KUKA KRL program: PPR-top-01.src

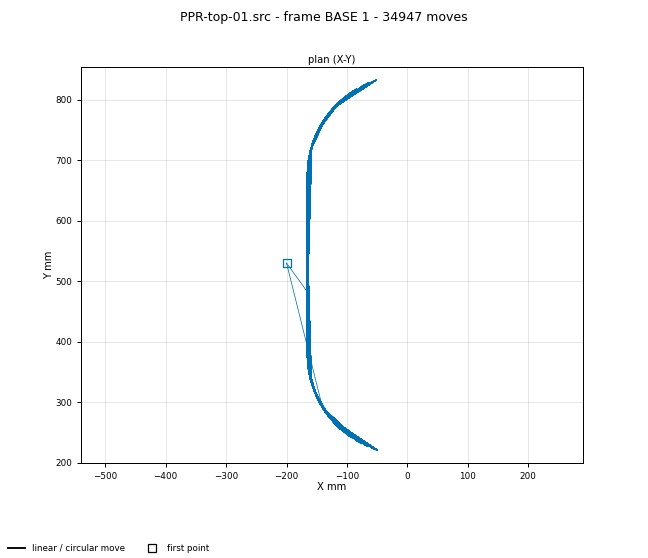
[picture p0: tool path of PPR-top-01.src in frame BASE 1, 34947 of 34948 moves have a stored position in this frame; points joined in program order, loops and branches not executed]
&ACCESS RVEO
&REL 11
&PARAM TEMPLATE = C:\KRC\Roboter\Template\vorgabe
&PARAM EDITMASK = *
DEF variable_helical2( )
;FOLD INI
  ;FOLD BASISTECH INI
    GLOBAL INTERRUPT DECL 3 WHEN $STOPMESS==TRUE DO IR_STOPM ( )
    INTERRUPT ON 3
    BAS (#INITMOV,0 )
  ;ENDFOLD (BASISTECH INI)
 ;FOLD USER INI


    ;Make your modifications here
  ;ENDFOLD (USER INI)
;ENDFOLD (INI)
ACTION(#AXIS_RESET,34,1000,#NOERROR,ERROR_CODE)
;FOLD PTP HOME  Vel= 100 % DEFAULT;%{PE}%MKUKATPBASIS,%CMOVE,%VPTP,%P 1:PTP, 2:HOME, 3:, 5:100, 7:DEFAULT
$BWDSTART = FALSE
PDAT_ACT=PDEFAULT
FDAT_ACT=FHOME
BAS (#PTP_PARAMS,100 )
$H_POS=XHOME
PTP  XHOME
;ENDFOLD
BAS(#TOOL,1)
BAS(#BASE,1)
$VEL_AXIS[1]=100
$VEL_AXIS[2]=100
$VEL_AXIS[3]=100
$VEL_AXIS[4]=100
$VEL_AXIS[5]=100
$VEL_AXIS[6]=100
$VEL_EXTAX[1]=100
$VEL_EXTAX[2]=100

$ACC_AXIS[1]=100
$ACC_AXIS[2]=100
$ACC_AXIS[3]=100
$ACC_AXIS[4]=100
$ACC_AXIS[5]=100
$ACC_AXIS[6]=100
$ACC_EXTAX[1]=100
$ACC_EXTAX[2]=100

;;;;;;;;; postprocessing parameters (date 2024-01-25T18:15:35.064605)
; qxconst: -165.65
; qxconstarcys: -151.5,145.5
; qE3offset: 0.00
; qyoffset: 530.00
; qswitchsplit: 3
; qthinningtol: 0.2010
;;;;;;;;;

SLIN {X  -200.000, Y  +530.000, Z    +0.000, A    +0.000, E1    +0.000, E3    +0.000, E4    +0.000}

SLIN {X  -140.419, Y  +290.622, Z    +0.000, E1   +73.705, E3  +372.898}
HALT
SPLINE
SPL {X  -135.839, Y  +283.697, Z    +0.000, E1   +73.388, E3  +378.636}
SPL {X  -131.903, Y  +278.292, Z    +0.000, E1   +73.096, E3  +383.125}
SPL {X  -129.007, Y  +274.590, Z    +0.000, E1   +72.484, E3  +388.421}
SPL {X  -124.646, Y  +269.397, Z    +0.000, E1   +72.041, E3  +393.170}
SPL {X  -111.023, Y  +255.562, Z    +0.000, E1   +75.772, E3  +384.951}
SPL {X   -49.289, Y  +220.353, Z    +0.000, E1   +56.690, E3  +577.666}
ENDSPLINE

SPLINE
SPL {X  -127.117, Y  +272.287, Z    +0.000, E1   +62.713, E3  +746.888}
SPL {X  -152.442, Y  +313.682, Z    +0.000, E1   +51.943, E3  +751.120}
SPL {X  -159.925, Y  +335.326, Z    +0.000, E1   +41.361, E3  +751.062}
SPL {X  -163.450, Y  +351.595, Z    +0.000, E1   +29.785, E3  +750.173}
SPL {X  -165.127, Y  +365.342, Z    +0.000, E1   +17.250, E3  +750.153}
SPL {X  -165.640, Y  +376.693, Z    +0.000, E1    +4.721, E3  +749.726}
SPL {X  -165.650, Y  +380.500, Z    +0.000, E1    -0.000, E3  +748.877}
SPL {X  -165.650, Y  +382.123, Z    +0.000, E1    -3.912, E3  +748.504}
SPL {X  -165.650, Y  +387.069, Z    +0.000, E1   -17.420, E3  +748.216}
SPL {X  -165.650, Y  +393.439, Z    +0.000, E1   -35.398, E3  +747.762}
SPL {X  -165.650, Y  +400.610, Z    +0.000, E1   -50.510, E3  +747.499}
SPL {X  -165.650, Y  +414.376, Z    +0.000, E1   -68.098, E3  +745.533}
SPL {X  -165.650, Y  +468.582, Z    +0.000, E1   -78.237, E3  +754.303}
SPL {X  -160.244, Y  +717.475, Z    +0.000, E1   -78.917, E3  +826.861}
SPL {X  -159.651, Y  +719.676, Z    +0.000, E1   -75.661, E3  +863.248}
SPL {X  -157.156, Y  +727.862, Z    +0.000, E1   -75.175, E3  +872.730}
SPL {X  -152.814, Y  +739.436, Z    +0.000, E1   -74.813, E3  +882.583}
SPL {X  -148.754, Y  +748.385, Z    +0.000, E1   -74.281, E3  +892.026}
SPL {X  -144.163, Y  +757.090, Z    +0.000, E1   -74.033, E3  +898.685}
SPL {X  -140.473, Y  +763.291, Z    +0.000, E1   -73.478, E3  +906.126}
SPL {X  -135.914, Y  +770.196, Z    +0.000, E1   -72.974, E3  +913.302}
SPL {X  -131.459, Y  +776.289, Z    +0.000, E1   -72.475, E3  +919.378}
SPL {X  -128.771, Y  +779.702, Z    +0.000, E1   -71.875, E3  +924.325}
SPL {X  -125.267, Y  +783.889, Z    +0.000, E1   -71.674, E3  +927.437}
SPL {X  -119.086, Y  +790.645, Z    +0.000, E1   -72.931, E3  +925.724}
SPL {X   -51.449, Y  +832.958, Z    +0.000, E1   -57.230, E3 +1083.244}
ENDSPLINE

SPLINE
SPL {X  -123.821, Y  +785.537, Z    +0.000, E1   -64.536, E3 +1284.989}
SPL {X  -153.467, Y  +737.853, Z    +0.000, E1   -51.757, E3 +1287.304}
SPL {X  -161.000, Y  +714.475, Z    +0.000, E1   -39.424, E3 +1286.776}
SPL {X  -164.534, Y  +694.695, Z    +0.000, E1   -23.511, E3 +1285.066}
SPL {X  -165.597, Y  +679.703, Z    +0.000, E1    -7.645, E3 +1284.942}
SPL {X  -165.650, Y  +673.520, Z    +0.000, E1    -0.048, E3 +1283.894}
SPL {X  -165.650, Y  +671.692, Z    +0.000, E1    +4.450, E3 +1283.460}
SPL {X  -165.650, Y  +667.743, Z    +0.000, E1   +15.617, E3 +1283.378}
SPL {X  -165.650, Y  +662.891, Z    +0.000, E1   +29.740, E3 +1282.896}
SPL {X  -165.650, Y  +655.319, Z    +0.000, E1   +47.265, E3 +1282.745}
SPL {X  -165.650, Y  +642.000, Z    +0.000, E1   +65.561, E3 +1281.726}
SPL {X  -165.650, Y  +619.979, Z    +0.000, E1   +79.465, E3 +1277.733}
SPL {X  -165.650, Y  +569.632, Z    +0.000, E1   +78.783, E3 +1293.011}
SPL {X  -158.840, Y  +331.491, Z    +0.000, E1   +77.462, E3 +1379.322}
ENDSPLINE

SPLINE
SPL {X  -159.893, Y  +335.208, Z    +0.000, E1   +75.483, E3 +1400.056}
ENDSPLINE

SPLINE
SPL {X  -156.487, Y  +324.170, Z    +0.000, E1   +75.150, E3 +1409.437}
SPL {X  -142.256, Y  +293.629, Z    +0.000, E1   +77.020, E3 +1404.537}
ENDSPLINE

SPLINE
SPL {X  -142.811, Y  +294.566, Z    +0.000, E1   +75.668, E3 +1416.499}
ENDSPLINE

SPLINE
SPL {X  -141.646, Y  +292.615, Z    +0.000, E1   +74.702, E3 +1425.593}
SPL {X  -140.419, Y  +290.622, Z    +0.000, E1   +73.705, E3 +1434.436}
SPL {X  -135.839, Y  +283.697, Z    +0.000, E1   +73.388, E3 +1440.174}
SPL {X  -131.336, Y  +277.551, Z    +0.000, E1   +72.879, E3 +1446.427}
SPL {X  -126.848, Y  +271.966, Z    +0.000, E1   +72.322, E3 +1452.155}
SPL {X  -123.729, Y  +268.359, Z    +0.000, E1   +71.932, E3 +1455.624}
SPL {X  -111.023, Y  +255.562, Z    +0.000, E1   +75.772, E3 +1446.490}
SPL {X   -52.752, Y  +221.474, Z    +0.000, E1   +59.157, E3 +1575.741}
SPL {X   -49.901, Y  +220.545, Z    +0.000, E1   +56.696, E3 +1662.134}
ENDSPLINE

SPLINE
SPL {X  -127.117, Y  +272.287, Z    +0.000, E1   +62.713, E3 +1808.427}
SPL {X  -152.442, Y  +313.682, Z    +0.000, E1   +51.943, E3 +1812.658}
SPL {X  -162.319, Y  +345.447, Z    +0.000, E1   +34.671, E3 +1812.084}
SPL {X  -165.127, Y  +365.342, Z    +0.000, E1   +17.250, E3 +1811.692}
SPL {X  -165.640, Y  +376.693, Z    +0.000, E1    +4.721, E3 +1811.265}
SPL {X  -165.650, Y  +380.500, Z    +0.000, E1    -0.000, E3 +1810.416}
SPL {X  -165.650, Y  +383.262, Z    +0.000, E1    -6.645, E3 +1809.945}
SPL {X  -165.650, Y  +388.390, Z    +0.000, E1   -21.508, E3 +1809.733}
SPL {X  -165.650, Y  +393.439, Z    +0.000, E1   -35.398, E3 +1809.300}
SPL {X  -165.650, Y  +400.610, Z    +0.000, E1   -50.510, E3 +1809.038}
SPL {X  -165.650, Y  +414.376, Z    +0.000, E1   -68.098, E3 +1807.071}
SPL {X  -165.650, Y  +468.582, Z    +0.000, E1   -78.237, E3 +1815.841}
SPL {X  -158.306, Y  +724.277, Z    +0.000, E1   -77.461, E3 +1906.283}
ENDSPLINE

SPLINE
SPL {X  -160.145, Y  +717.851, Z    +0.000, E1   -75.386, E3 +1926.796}
ENDSPLINE

SPLINE
SPL {X  -157.156, Y  +727.862, Z    +0.000, E1   -75.175, E3 +1934.268}
SPL {X  -154.068, Y  +736.353, Z    +0.000, E1   -74.906, E3 +1941.443}
SPL {X  -149.738, Y  +746.340, Z    +0.000, E1   -74.451, E3 +1951.131}
SPL {X  -144.163, Y  +757.090, Z    +0.000, E1   -74.033, E3 +1960.223}
SPL {X  -139.284, Y  +765.165, Z    +0.000, E1   -73.322, E3 +1969.918}
SPL {X  -134.662, Y  +771.969, Z    +0.000, E1   -72.884, E3 +1976.249}
SPL {X  -131.459, Y  +776.289, Z    +0.000, E1   -72.475, E3 +1980.917}
SPL {X  -127.605, Y  +781.126, Z    +0.000, E1   -71.922, E3 +1986.361}
SPL {X  -124.773, Y  +784.457, Z    +0.000, E1   -71.383, E3 +1990.408}
SPL {X  -119.086, Y  +790.645, Z    +0.000, E1   -72.931, E3 +1987.262}
SPL {X   -54.274, Y  +832.006, Z    +0.000, E1   -58.502, E3 +2117.475}
SPL {X   -50.797, Y  +833.169, Z    +0.000, E1   -57.000, E3 +2212.824}
ENDSPLINE

SPLINE
SPL {X  -113.713, Y  +795.955, Z    +0.000, E1   -65.735, E3 +2343.701}
SPL {X  -131.116, Y  +776.736, Z    +0.000, E1   -63.149, E3 +2348.231}
SPL {X  -153.467, Y  +737.853, Z    +0.000, E1   -51.757, E3 +2348.842}
SPL {X  -162.176, Y  +709.248, Z    +0.000, E1   -35.773, E3 +2347.868}
SPL {X  -164.888, Y  +691.368, Z    +0.000, E1   -20.174, E3 +2346.305}
SPL {X  -165.597, Y  +679.703, Z    +0.000, E1    -7.645, E3 +2346.480}
SPL {X  -165.650, Y  +673.520, Z    +0.000, E1    -0.048, E3 +2345.432}
SPL {X  -165.650, Y  +671.692, Z    +0.000, E1    +4.450, E3 +2344.999}
SPL {X  -165.650, Y  +667.743, Z    +0.000, E1   +15.617, E3 +2344.917}
SPL {X  -165.650, Y  +662.891, Z    +0.000, E1   +29.740, E3 +2344.434}
SPL {X  -165.650, Y  +658.373, Z    +0.000, E1   +40.877, E3 +2344.632}
SPL {X  -165.650, Y  +650.834, Z    +0.000, E1   +55.143, E3 +2343.885}
SPL {X  -165.650, Y  +639.785, Z    +0.000, E1   +67.512, E3 +2343.102}
SPL {X  -165.650, Y  +619.979, Z    +0.000, E1   +79.465, E3 +2339.271}
SPL {X  -165.650, Y  +584.722, Z    +0.000, E1   +79.551, E3 +2348.562}
SPL {X  -165.650, Y  +560.326, Z    +0.000, E1   +78.360, E3 +2358.284}
SPL {X  -160.258, Y  +336.579, Z    +0.000, E1   +78.314, E3 +2429.806}
SPL {X  -159.618, Y  +334.207, Z    +0.000, E1   +75.622, E3 +2460.620}
SPL {X  -156.487, Y  +324.170, Z    +0.000, E1   +75.150, E3 +2470.976}
SPL {X  -142.256, Y  +293.629, Z    +0.000, E1   +77.020, E3 +2466.076}
ENDSPLINE

SPLINE
SPL {X  -142.811, Y  +294.566, Z    +0.000, E1   +75.668, E3 +2478.038}
ENDSPLINE

SPLINE
SPL {X  -141.646, Y  +292.615, Z    +0.000, E1   +74.702, E3 +2487.131}
SPL {X  -140.419, Y  +290.622, Z    +0.000, E1   +73.705, E3 +2495.975}
SPL {X  -136.008, Y  +283.940, Z    +0.000, E1   +73.594, E3 +2500.094}
SPL {X  -132.748, Y  +279.415, Z    +0.000, E1   +73.006, E3 +2506.150}
SPL {X  -129.007, Y  +274.590, Z    +0.000, E1   +72.484, E3 +2511.498}
SPL {X  -125.914, Y  +270.864, Z    +0.000, E1   +72.144, E3 +2514.990}
SPL {X  -123.729, Y  +268.359, Z    +0.000, E1   +71.932, E3 +2517.162}
SPL {X  -111.023, Y  +255.562, Z    +0.000, E1   +75.772, E3 +2508.028}
SPL {X   -49.289, Y  +220.353, Z    +0.000, E1   +56.690, E3 +2700.743}
ENDSPLINE

SPLINE
SPL {X  -127.117, Y  +272.287, Z    +0.000, E1   +62.713, E3 +2869.965}
SPL {X  -154.956, Y  +319.945, Z    +0.000, E1   +49.402, E3 +2874.364}
SPL {X  -162.871, Y  +348.286, Z    +0.000, E1   +32.462, E3 +2873.392}
SPL {X  -165.127, Y  +365.342, Z    +0.000, E1   +17.250, E3 +2873.230}
SPL {X  -165.640, Y  +376.693, Z    +0.000, E1    +4.721, E3 +2872.803}
SPL {X  -165.650, Y  +380.500, Z    +0.000, E1    -0.000, E3 +2871.954}
SPL {X  -165.650, Y  +382.123, Z    +0.000, E1    -3.912, E3 +2871.581}
SPL {X  -165.650, Y  +387.069, Z    +0.000, E1   -17.420, E3 +2871.293}
SPL {X  -165.650, Y  +393.439, Z    +0.000, E1   -35.398, E3 +2870.839}
SPL {X  -165.650, Y  +400.610, Z    +0.000, E1   -50.510, E3 +2870.576}
SPL {X  -165.650, Y  +414.376, Z    +0.000, E1   -68.098, E3 +2868.610}
SPL {X  -165.650, Y  +468.582, Z    +0.000, E1   -78.237, E3 +2877.380}
SPL {X  -160.244, Y  +717.475, Z    +0.000, E1   -78.917, E3 +2949.938}
SPL {X  -159.651, Y  +719.676, Z    +0.000, E1   -75.661, E3 +2986.324}
SPL {X  -157.156, Y  +727.862, Z    +0.000, E1   -75.175, E3 +2995.807}
SPL {X  -154.068, Y  +736.353, Z    +0.000, E1   -74.906, E3 +3002.981}
SPL {X  -149.738, Y  +746.340, Z    +0.000, E1   -74.451, E3 +3012.669}
SPL {X  -144.163, Y  +757.090, Z    +0.000, E1   -74.033, E3 +3021.762}
SPL {X  -139.284, Y  +765.165, Z    +0.000, E1   -73.322, E3 +3031.456}
SPL {X  -134.662, Y  +771.969, Z    +0.000, E1   -72.884, E3 +3037.788}
SPL {X  -131.459, Y  +776.289, Z    +0.000, E1   -72.475, E3 +3042.455}
SPL {X  -127.605, Y  +781.126, Z    +0.000, E1   -71.922, E3 +3047.899}
SPL {X  -124.773, Y  +784.457, Z    +0.000, E1   -71.383, E3 +3051.947}
SPL {X  -119.086, Y  +790.645, Z    +0.000, E1   -72.931, E3 +3048.801}
SPL {X   -51.449, Y  +832.958, Z    +0.000, E1   -57.230, E3 +3206.321}
ENDSPLINE

SPLINE
SPL {X  -123.821, Y  +785.537, Z    +0.000, E1   -64.536, E3 +3408.066}
SPL {X  -153.467, Y  +737.853, Z    +0.000, E1   -51.757, E3 +3410.381}
SPL {X  -161.000, Y  +714.475, Z    +0.000, E1   -39.424, E3 +3409.853}
SPL {X  -164.534, Y  +694.695, Z    +0.000, E1   -23.511, E3 +3408.143}
SPL {X  -165.597, Y  +679.703, Z    +0.000, E1    -7.645, E3 +3408.019}
SPL {X  -165.650, Y  +673.520, Z    +0.000, E1    -0.048, E3 +3406.971}
SPL {X  -165.650, Y  +671.692, Z    +0.000, E1    +4.450, E3 +3406.537}
SPL {X  -165.650, Y  +667.743, Z    +0.000, E1   +15.617, E3 +3406.455}
SPL {X  -165.650, Y  +661.459, Z    +0.000, E1   +33.218, E3 +3406.035}
SPL {X  -165.650, Y  +653.296, Z    +0.000, E1   +51.333, E3 +3405.591}
SPL {X  -165.650, Y  +642.000, Z    +0.000, E1   +65.561, E3 +3404.803}
SPL {X  -165.650, Y  +619.979, Z    +0.000, E1   +79.465, E3 +3400.810}
SPL {X  -165.650, Y  +569.632, Z    +0.000, E1   +78.783, E3 +3416.088}
SPL {X  -158.840, Y  +331.491, Z    +0.000, E1   +77.462, E3 +3502.398}
ENDSPLINE

SPLINE
SPL {X  -159.893, Y  +335.208, Z    +0.000, E1   +75.483, E3 +3523.133}
ENDSPLINE

SPLINE
SPL {X  -156.487, Y  +324.170, Z    +0.000, E1   +75.150, E3 +3532.514}
SPL {X  -142.256, Y  +293.629, Z    +0.000, E1   +77.020, E3 +3527.614}
ENDSPLINE

SPLINE
SPL {X  -142.811, Y  +294.566, Z    +0.000, E1   +75.668, E3 +3539.576}
ENDSPLINE

SPLINE
SPL {X  -141.646, Y  +292.615, Z    +0.000, E1   +74.702, E3 +3548.670}
SPL {X  -140.419, Y  +290.622, Z    +0.000, E1   +73.705, E3 +3557.513}
SPL {X  -136.008, Y  +283.940, Z    +0.000, E1   +73.594, E3 +3561.632}
SPL {X  -132.748, Y  +279.415, Z    +0.000, E1   +73.006, E3 +3567.688}
SPL {X  -129.007, Y  +274.590, Z    +0.000, E1   +72.484, E3 +3573.037}
SPL {X  -125.914, Y  +270.864, Z    +0.000, E1   +72.144, E3 +3576.528}
SPL {X  -123.729, Y  +268.359, Z    +0.000, E1   +71.932, E3 +3578.701}
SPL {X  -111.023, Y  +255.562, Z    +0.000, E1   +75.772, E3 +3569.567}
SPL {X   -49.289, Y  +220.353, Z    +0.000, E1   +56.690, E3 +3762.282}
ENDSPLINE

SPLINE
SPL {X  -127.117, Y  +272.287, Z    +0.000, E1   +62.713, E3 +3931.503}
SPL {X  -154.956, Y  +319.945, Z    +0.000, E1   +49.402, E3 +3935.903}
SPL {X  -162.871, Y  +348.286, Z    +0.000, E1   +32.462, E3 +3934.930}
SPL {X  -165.127, Y  +365.342, Z    +0.000, E1   +17.250, E3 +3934.769}
SPL {X  -165.640, Y  +376.693, Z    +0.000, E1    +4.721, E3 +3934.342}
SPL {X  -165.650, Y  +380.500, Z    +0.000, E1    -0.000, E3 +3933.493}
SPL {X  -165.650, Y  +383.262, Z    +0.000, E1    -6.645, E3 +3933.022}
SPL {X  -165.650, Y  +388.390, Z    +0.000, E1   -21.508, E3 +3932.809}
SPL {X  -165.650, Y  +393.439, Z    +0.000, E1   -35.398, E3 +3932.377}
SPL {X  -165.650, Y  +400.610, Z    +0.000, E1   -50.510, E3 +3932.115}
SPL {X  -165.650, Y  +414.376, Z    +0.000, E1   -68.098, E3 +3930.148}
SPL {X  -165.650, Y  +468.582, Z    +0.000, E1   -78.237, E3 +3938.918}
SPL {X  -158.306, Y  +724.277, Z    +0.000, E1   -77.461, E3 +4029.360}
ENDSPLINE

SPLINE
SPL {X  -160.145, Y  +717.851, Z    +0.000, E1   -75.386, E3 +4049.873}
ENDSPLINE

SPLINE
SPL {X  -157.156, Y  +727.862, Z    +0.000, E1   -75.175, E3 +4057.345}
SPL {X  -154.068, Y  +736.353, Z    +0.000, E1   -74.906, E3 +4064.520}
SPL {X  -149.738, Y  +746.340, Z    +0.000, E1   -74.451, E3 +4074.208}
SPL {X  -144.163, Y  +757.090, Z    +0.000, E1   -74.033, E3 +4083.300}
SPL {X  -139.284, Y  +765.165, Z    +0.000, E1   -73.322, E3 +4092.995}
SPL {X  -134.662, Y  +771.969, Z    +0.000, E1   -72.884, E3 +4099.326}
SPL {X  -131.459, Y  +776.289, Z    +0.000, E1   -72.475, E3 +4103.994}
SPL {X  -127.605, Y  +781.126, Z    +0.000, E1   -71.922, E3 +4109.438}
SPL {X  -124.773, Y  +784.457, Z    +0.000, E1   -71.383, E3 +4113.485}
SPL {X  -119.086, Y  +790.645, Z    +0.000, E1   -72.931, E3 +4110.339}
SPL {X   -51.449, Y  +832.958, Z    +0.000, E1   -57.230, E3 +4267.859}
ENDSPLINE

SPLINE
SPL {X  -123.821, Y  +785.537, Z    +0.000, E1   -64.536, E3 +4469.604}
SPL {X  -153.467, Y  +737.853, Z    +0.000, E1   -51.757, E3 +4471.919}
SPL {X  -161.000, Y  +714.475, Z    +0.000, E1   -39.424, E3 +4471.392}
SPL {X  -164.534, Y  +694.695, Z    +0.000, E1   -23.511, E3 +4469.682}
SPL {X  -165.597, Y  +679.703, Z    +0.000, E1    -7.645, E3 +4469.557}
SPL {X  -165.650, Y  +673.520, Z    +0.000, E1    -0.048, E3 +4468.509}
SPL {X  -165.650, Y  +671.692, Z    +0.000, E1    +4.450, E3 +4468.076}
SPL {X  -165.650, Y  +667.743, Z    +0.000, E1   +15.617, E3 +4467.994}
SPL {X  -165.650, Y  +661.459, Z    +0.000, E1   +33.218, E3 +4467.574}
SPL {X  -165.650, Y  +653.296, Z    +0.000, E1   +51.333, E3 +4467.129}
SPL {X  -165.650, Y  +642.000, Z    +0.000, E1   +65.561, E3 +4466.341}
SPL {X  -165.650, Y  +619.979, Z    +0.000, E1   +79.465, E3 +4462.348}
SPL {X  -165.650, Y  +569.632, Z    +0.000, E1   +78.783, E3 +4477.627}
SPL {X  -158.840, Y  +331.491, Z    +0.000, E1   +77.462, E3 +4563.937}
ENDSPLINE

SPLINE
SPL {X  -159.893, Y  +335.208, Z    +0.000, E1   +75.483, E3 +4584.672}
ENDSPLINE

SPLINE
SPL {X  -156.487, Y  +324.170, Z    +0.000, E1   +75.150, E3 +4594.053}
SPL {X  -142.256, Y  +293.629, Z    +0.000, E1   +77.020, E3 +4589.152}
ENDSPLINE

SPLINE
SPL {X  -142.811, Y  +294.566, Z    +0.000, E1   +75.668, E3 +4601.115}
ENDSPLINE

SPLINE
SPL {X  -141.646, Y  +292.615, Z    +0.000, E1   +74.702, E3 +4610.208}
SPL {X  -140.419, Y  +290.622, Z    +0.000, E1   +73.705, E3 +4619.052}
SPL {X  -136.008, Y  +283.940, Z    +0.000, E1   +73.594, E3 +4623.171}
SPL {X  -132.748, Y  +279.415, Z    +0.000, E1   +73.006, E3 +4629.226}
SPL {X  -129.007, Y  +274.590, Z    +0.000, E1   +72.484, E3 +4634.575}
SPL {X  -125.914, Y  +270.864, Z    +0.000, E1   +72.144, E3 +4638.067}
SPL {X  -123.729, Y  +268.359, Z    +0.000, E1   +71.932, E3 +4640.239}
SPL {X  -111.023, Y  +255.562, Z    +0.000, E1   +75.772, E3 +4631.105}
SPL {X   -49.289, Y  +220.353, Z    +0.000, E1   +56.690, E3 +4823.820}
ENDSPLINE

SPLINE
SPL {X  -127.117, Y  +272.287, Z    +0.000, E1   +62.713, E3 +4993.042}
SPL {X  -154.956, Y  +319.945, Z    +0.000, E1   +49.402, E3 +4997.441}
SPL {X  -162.871, Y  +348.286, Z    +0.000, E1   +32.462, E3 +4996.469}
SPL {X  -165.127, Y  +365.342, Z    +0.000, E1   +17.250, E3 +4996.307}
SPL {X  -165.640, Y  +376.693, Z    +0.000, E1    +4.721, E3 +4995.880}
SPL {X  -165.650, Y  +380.500, Z    +0.000, E1    -0.000, E3 +4995.031}
SPL {X  -165.650, Y  +383.262, Z    +0.000, E1    -6.645, E3 +4994.560}
SPL {X  -165.650, Y  +388.390, Z    +0.000, E1   -21.508, E3 +4994.348}
SPL {X  -165.650, Y  +393.439, Z    +0.000, E1   -35.398, E3 +4993.915}
SPL {X  -165.650, Y  +400.610, Z    +0.000, E1   -50.510, E3 +4993.653}
SPL {X  -165.650, Y  +414.376, Z    +0.000, E1   -68.098, E3 +4991.687}
SPL {X  -165.650, Y  +468.582, Z    +0.000, E1   -78.237, E3 +5000.457}
SPL {X  -158.306, Y  +724.277, Z    +0.000, E1   -77.461, E3 +5090.898}
ENDSPLINE

SPLINE
SPL {X  -160.145, Y  +717.851, Z    +0.000, E1   -75.386, E3 +5111.412}
ENDSPLINE

SPLINE
SPL {X  -157.156, Y  +727.862, Z    +0.000, E1   -75.175, E3 +5118.884}
SPL {X  -154.068, Y  +736.353, Z    +0.000, E1   -74.906, E3 +5126.058}
SPL {X  -149.738, Y  +746.340, Z    +0.000, E1   -74.451, E3 +5135.746}
SPL {X  -144.163, Y  +757.090, Z    +0.000, E1   -74.033, E3 +5144.838}
SPL {X  -139.284, Y  +765.165, Z    +0.000, E1   -73.322, E3 +5154.533}
SPL {X  -134.662, Y  +771.969, Z    +0.000, E1   -72.884, E3 +5160.865}
SPL {X  -131.459, Y  +776.289, Z    +0.000, E1   -72.475, E3 +5165.532}
SPL {X  -127.605, Y  +781.126, Z    +0.000, E1   -71.922, E3 +5170.976}
SPL {X  -124.773, Y  +784.457, Z    +0.000, E1   -71.383, E3 +5175.024}
SPL {X  -119.086, Y  +790.645, Z    +0.000, E1   -72.931, E3 +5171.878}
SPL {X   -51.449, Y  +832.958, Z    +0.000, E1   -57.230, E3 +5329.398}
ENDSPLINE

SPLINE
SPL {X  -123.821, Y  +785.537, Z    +0.000, E1   -64.536, E3 +5531.143}
SPL {X  -153.467, Y  +737.853, Z    +0.000, E1   -51.757, E3 +5533.458}
SPL {X  -161.000, Y  +714.475, Z    +0.000, E1   -39.424, E3 +5532.930}
SPL {X  -164.534, Y  +694.695, Z    +0.000, E1   -23.511, E3 +5531.220}
SPL {X  -165.597, Y  +679.703, Z    +0.000, E1    -7.645, E3 +5531.096}
SPL {X  -165.650, Y  +673.520, Z    +0.000, E1    -0.048, E3 +5530.048}
SPL {X  -165.650, Y  +671.692, Z    +0.000, E1    +4.450, E3 +5529.614}
SPL {X  -165.650, Y  +667.743, Z    +0.000, E1   +15.617, E3 +5529.532}
SPL {X  -165.650, Y  +661.459, Z    +0.000, E1   +33.218, E3 +5529.112}
SPL {X  -165.650, Y  +653.296, Z    +0.000, E1   +51.333, E3 +5528.668}
SPL {X  -165.650, Y  +642.000, Z    +0.000, E1   +65.561, E3 +5527.880}
SPL {X  -165.650, Y  +619.979, Z    +0.000, E1   +79.465, E3 +5523.886}
SPL {X  -165.650, Y  +569.632, Z    +0.000, E1   +78.783, E3 +5539.165}
SPL {X  -158.840, Y  +331.491, Z    +0.000, E1   +77.462, E3 +5625.475}
ENDSPLINE

SPLINE
SPL {X  -159.893, Y  +335.208, Z    +0.000, E1   +75.483, E3 +5646.210}
ENDSPLINE

SPLINE
SPL {X  -156.487, Y  +324.170, Z    +0.000, E1   +75.150, E3 +5655.591}
SPL {X  -142.256, Y  +293.629, Z    +0.000, E1   +77.020, E3 +5650.691}
ENDSPLINE

SPLINE
SPL {X  -142.811, Y  +294.566, Z    +0.000, E1   +75.668, E3 +5662.653}
ENDSPLINE

SPLINE
SPL {X  -141.646, Y  +292.615, Z    +0.000, E1   +74.702, E3 +5671.747}
SPL {X  -140.419, Y  +290.622, Z    +0.000, E1   +73.705, E3 +5680.590}
SPL {X  -136.008, Y  +283.940, Z    +0.000, E1   +73.594, E3 +5684.709}
SPL {X  -132.748, Y  +279.415, Z    +0.000, E1   +73.006, E3 +5690.765}
SPL {X  -129.007, Y  +274.590, Z    +0.000, E1   +72.484, E3 +5696.114}
SPL {X  -125.914, Y  +270.864, Z    +0.000, E1   +72.144, E3 +5699.605}
SPL {X  -123.729, Y  +268.359, Z    +0.000, E1   +71.932, E3 +5701.778}
SPL {X  -111.023, Y  +255.562, Z    +0.000, E1   +75.772, E3 +5692.644}
SPL {X   -49.289, Y  +220.353, Z    +0.000, E1   +56.690, E3 +5885.358}
ENDSPLINE

SPLINE
SPL {X  -127.117, Y  +272.287, Z    +0.000, E1   +62.713, E3 +6054.580}
SPL {X  -154.956, Y  +319.945, Z    +0.000, E1   +49.402, E3 +6058.979}
SPL {X  -162.871, Y  +348.286, Z    +0.000, E1   +32.462, E3 +6058.007}
SPL {X  -165.127, Y  +365.342, Z    +0.000, E1   +17.250, E3 +6057.846}
SPL {X  -165.640, Y  +376.693, Z    +0.000, E1    +4.721, E3 +6057.419}
SPL {X  -165.650, Y  +380.500, Z    +0.000, E1    -0.000, E3 +6056.569}
SPL {X  -165.650, Y  +382.123, Z    +0.000, E1    -3.912, E3 +6056.197}
SPL {X  -165.650, Y  +387.069, Z    +0.000, E1   -17.420, E3 +6055.908}
SPL {X  -165.650, Y  +393.439, Z    +0.000, E1   -35.398, E3 +6055.454}
SPL {X  -165.650, Y  +402.896, Z    +0.000, E1   -54.480, E3 +6054.695}
SPL {X  -165.650, Y  +416.934, Z    +0.000, E1   -69.887, E3 +6053.161}
SPL {X  -165.650, Y  +459.729, Z    +0.000, E1   -78.035, E3 +6059.680}
SPL {X  -165.650, Y  +475.450, Z    +0.000, E1   -78.345, E3 +6063.794}
SPL {X  -160.244, Y  +717.475, Z    +0.000, E1   -78.917, E3 +6134.553}
SPL {X  -159.651, Y  +719.676, Z    +0.000, E1   -75.661, E3 +6170.940}
SPL {X  -157.156, Y  +727.862, Z    +0.000, E1   -75.175, E3 +6180.422}
SPL {X  -154.068, Y  +736.353, Z    +0.000, E1   -74.906, E3 +6187.597}
SPL {X  -149.738, Y  +746.340, Z    +0.000, E1   -74.451, E3 +6197.284}
SPL {X  -144.163, Y  +757.090, Z    +0.000, E1   -74.033, E3 +6206.377}
SPL {X  -139.284, Y  +765.165, Z    +0.000, E1   -73.322, E3 +6216.072}
SPL {X  -134.662, Y  +771.969, Z    +0.000, E1   -72.884, E3 +6222.403}
SPL {X  -131.459, Y  +776.289, Z    +0.000, E1   -72.475, E3 +6227.070}
SPL {X  -128.771, Y  +779.702, Z    +0.000, E1   -71.875, E3 +6232.017}
SPL {X  -125.267, Y  +783.889, Z    +0.000, E1   -71.674, E3 +6235.129}
SPL {X  -119.086, Y  +790.645, Z    +0.000, E1   -72.931, E3 +6233.416}
SPL {X   -51.449, Y  +832.958, Z    +0.000, E1   -57.230, E3 +6390.936}
ENDSPLINE

SPLINE
SPL {X  -123.821, Y  +785.537, Z    +0.000, E1   -64.536, E3 +6592.681}
SPL {X  -153.467, Y  +737.853, Z    +0.000, E1   -51.757, E3 +6594.996}
SPL {X  -162.176, Y  +709.248, Z    +0.000, E1   -35.773, E3 +6594.022}
SPL {X  -164.888, Y  +691.368, Z    +0.000, E1   -20.174, E3 +6592.459}
SPL {X  -165.597, Y  +679.703, Z    +0.000, E1    -7.645, E3 +6592.634}
SPL {X  -165.650, Y  +673.520, Z    +0.000, E1    -0.048, E3 +6591.586}
SPL {X  -165.650, Y  +671.692, Z    +0.000, E1    +4.450, E3 +6591.153}
SPL {X  -165.650, Y  +667.743, Z    +0.000, E1   +15.617, E3 +6591.070}
SPL {X  -165.650, Y  +661.459, Z    +0.000, E1   +33.218, E3 +6590.651}
SPL {X  -165.650, Y  +653.296, Z    +0.000, E1   +51.333, E3 +6590.206}
SPL {X  -165.650, Y  +642.000, Z    +0.000, E1   +65.561, E3 +6589.418}
SPL {X  -165.650, Y  +619.979, Z    +0.000, E1   +79.465, E3 +6585.425}
SPL {X  -165.650, Y  +584.722, Z    +0.000, E1   +79.551, E3 +6594.716}
SPL {X  -165.650, Y  +560.326, Z    +0.000, E1   +78.360, E3 +6604.438}
SPL {X  -158.840, Y  +331.491, Z    +0.000, E1   +77.462, E3 +6687.014}
ENDSPLINE

SPLINE
SPL {X  -159.893, Y  +335.208, Z    +0.000, E1   +75.483, E3 +6707.748}
ENDSPLINE

SPLINE
SPL {X  -156.487, Y  +324.170, Z    +0.000, E1   +75.150, E3 +6717.130}
SPL {X  -142.256, Y  +293.629, Z    +0.000, E1   +77.020, E3 +6712.229}
ENDSPLINE

SPLINE
SPL {X  -142.811, Y  +294.566, Z    +0.000, E1   +75.668, E3 +6724.192}
ENDSPLINE

SPLINE
SPL {X  -141.646, Y  +292.615, Z    +0.000, E1   +74.702, E3 +6733.285}
SPL {X  -140.419, Y  +290.622, Z    +0.000, E1   +73.705, E3 +6742.129}
SPL {X  -136.008, Y  +283.940, Z    +0.000, E1   +73.594, E3 +6746.248}
SPL {X  -132.748, Y  +279.415, Z    +0.000, E1   +73.006, E3 +6752.303}
SPL {X  -129.007, Y  +274.590, Z    +0.000, E1   +72.484, E3 +6757.652}
SPL {X  -125.914, Y  +270.864, Z    +0.000, E1   +72.144, E3 +6761.144}
SPL {X  -123.729, Y  +268.359, Z    +0.000, E1   +71.932, E3 +6763.316}
SPL {X  -111.023, Y  +255.562, Z    +0.000, E1   +75.772, E3 +6754.182}
SPL {X   -49.289, Y  +220.353, Z    +0.000, E1   +56.690, E3 +6946.897}
ENDSPLINE

SPLINE
SPL {X  -127.117, Y  +272.287, Z    +0.000, E1   +62.713, E3 +7116.119}
SPL {X  -152.442, Y  +313.682, Z    +0.000, E1   +51.943, E3 +7120.351}
SPL {X  -159.925, Y  +335.326, Z    +0.000, E1   +41.361, E3 +7120.293}
SPL {X  -163.450, Y  +351.595, Z    +0.000, E1   +29.785, E3 +7119.404}
SPL {X  -165.127, Y  +365.342, Z    +0.000, E1   +17.250, E3 +7119.384}
SPL {X  -165.640, Y  +376.693, Z    +0.000, E1    +4.721, E3 +7118.957}
SPL {X  -165.650, Y  +380.500, Z    +0.000, E1    -0.000, E3 +7118.108}
SPL {X  -165.650, Y  +382.123, Z    +0.000, E1    -3.912, E3 +7117.735}
SPL {X  -165.650, Y  +387.069, Z    +0.000, E1   -17.420, E3 +7117.447}
SPL {X  -165.650, Y  +393.439, Z    +0.000, E1   -35.398, E3 +7116.992}
SPL {X  -165.650, Y  +400.610, Z    +0.000, E1   -50.510, E3 +7116.730}
SPL {X  -165.650, Y  +414.376, Z    +0.000, E1   -68.098, E3 +7114.764}
SPL {X  -165.650, Y  +468.582, Z    +0.000, E1   -78.237, E3 +7123.534}
SPL {X  -160.244, Y  +717.475, Z    +0.000, E1   -78.917, E3 +7196.092}
SPL {X  -159.651, Y  +719.676, Z    +0.000, E1   -75.661, E3 +7232.478}
SPL {X  -157.156, Y  +727.862, Z    +0.000, E1   -75.175, E3 +7241.961}
SPL {X  -152.814, Y  +739.436, Z    +0.000, E1   -74.813, E3 +7251.814}
SPL {X  -148.754, Y  +748.385, Z    +0.000, E1   -74.281, E3 +7261.256}
SPL {X  -144.163, Y  +757.090, Z    +0.000, E1   -74.033, E3 +7267.915}
SPL {X  -140.473, Y  +763.291, Z    +0.000, E1   -73.478, E3 +7275.357}
SPL {X  -135.914, Y  +770.196, Z    +0.000, E1   -72.974, E3 +7282.533}
SPL {X  -131.459, Y  +776.289, Z    +0.000, E1   -72.475, E3 +7288.609}
SPL {X  -128.771, Y  +779.702, Z    +0.000, E1   -71.875, E3 +7293.556}
SPL {X  -125.267, Y  +783.889, Z    +0.000, E1   -71.674, E3 +7296.668}
SPL {X  -119.086, Y  +790.645, Z    +0.000, E1   -72.931, E3 +7294.955}
SPL {X   -51.449, Y  +832.958, Z    +0.000, E1   -57.230, E3 +7452.475}
ENDSPLINE

SPLINE
SPL {X  -123.821, Y  +785.537, Z    +0.000, E1   -64.536, E3 +7654.220}
SPL {X  -153.467, Y  +737.853, Z    +0.000, E1   -51.757, E3 +7656.534}
SPL {X  -161.000, Y  +714.475, Z    +0.000, E1   -39.424, E3 +7656.007}
SPL {X  -164.534, Y  +694.695, Z    +0.000, E1   -23.511, E3 +7654.297}
SPL {X  -165.597, Y  +679.703, Z    +0.000, E1    -7.645, E3 +7654.173}
SPL {X  -165.650, Y  +673.520, Z    +0.000, E1    -0.048, E3 +7653.124}
SPL {X  -165.650, Y  +671.692, Z    +0.000, E1    +4.450, E3 +7652.691}
SPL {X  -165.650, Y  +667.743, Z    +0.000, E1   +15.617, E3 +7652.609}
SPL {X  -165.650, Y  +662.891, Z    +0.000, E1   +29.740, E3 +7652.127}
SPL {X  -165.650, Y  +655.319, Z    +0.000, E1   +47.265, E3 +7651.976}
SPL {X  -165.650, Y  +642.000, Z    +0.000, E1   +65.561, E3 +7650.957}
SPL {X  -165.650, Y  +619.979, Z    +0.000, E1   +79.465, E3 +7646.963}
SPL {X  -165.650, Y  +569.632, Z    +0.000, E1   +78.783, E3 +7662.242}
SPL {X  -158.840, Y  +331.491, Z    +0.000, E1   +77.462, E3 +7748.552}
ENDSPLINE

SPLINE
SPL {X  -159.893, Y  +335.208, Z    +0.000, E1   +75.483, E3 +7769.287}
ENDSPLINE

SPLINE
SPL {X  -156.487, Y  +324.170, Z    +0.000, E1   +75.150, E3 +7778.668}
SPL {X  -142.256, Y  +293.629, Z    +0.000, E1   +77.020, E3 +7773.768}
ENDSPLINE

SPLINE
SPL {X  -142.811, Y  +294.566, Z    +0.000, E1   +75.668, E3 +7785.730}
ENDSPLINE

SPLINE
SPL {X  -141.646, Y  +292.615, Z    +0.000, E1   +74.702, E3 +7794.824}
SPL {X  -140.419, Y  +290.622, Z    +0.000, E1   +73.705, E3 +7803.667}
SPL {X  -136.008, Y  +283.940, Z    +0.000, E1   +73.594, E3 +7807.786}
SPL {X  -132.748, Y  +279.415, Z    +0.000, E1   +73.006, E3 +7813.842}
SPL {X  -129.007, Y  +274.590, Z    +0.000, E1   +72.484, E3 +7819.191}
SPL {X  -125.914, Y  +270.864, Z    +0.000, E1   +72.144, E3 +7822.682}
SPL {X  -123.729, Y  +268.359, Z    +0.000, E1   +71.932, E3 +7824.855}
SPL {X  -111.023, Y  +255.562, Z    +0.000, E1   +75.772, E3 +7815.720}
SPL {X   -52.752, Y  +221.474, Z    +0.000, E1   +59.157, E3 +7944.972}
SPL {X   -49.901, Y  +220.545, Z    +0.000, E1   +56.696, E3 +8031.365}
ENDSPLINE

SPLINE
SPL {X  -127.117, Y  +272.287, Z    +0.000, E1   +62.713, E3 +8177.657}
SPL {X  -152.442, Y  +313.682, Z    +0.000, E1   +51.943, E3 +8181.889}
SPL {X  -162.319, Y  +345.447, Z    +0.000, E1   +34.671, E3 +8181.315}
SPL {X  -165.127, Y  +365.342, Z    +0.000, E1   +17.250, E3 +8180.923}
SPL {X  -165.640, Y  +376.693, Z    +0.000, E1    +4.721, E3 +8180.496}
SPL {X  -165.650, Y  +380.500, Z    +0.000, E1    -0.000, E3 +8179.646}
SPL {X  -165.650, Y  +382.123, Z    +0.000, E1    -3.912, E3 +8179.274}
SPL {X  -165.650, Y  +387.069, Z    +0.000, E1   -17.420, E3 +8178.985}
SPL {X  -165.650, Y  +393.439, Z    +0.000, E1   -35.398, E3 +8178.531}
SPL {X  -165.650, Y  +400.610, Z    +0.000, E1   -50.510, E3 +8178.268}
SPL {X  -165.650, Y  +414.376, Z    +0.000, E1   -68.098, E3 +8176.302}
SPL {X  -165.650, Y  +468.582, Z    +0.000, E1   -78.237, E3 +8185.072}
SPL {X  -160.244, Y  +717.475, Z    +0.000, E1   -78.917, E3 +8257.630}
SPL {X  -159.651, Y  +719.676, Z    +0.000, E1   -75.661, E3 +8294.017}
SPL {X  -157.156, Y  +727.862, Z    +0.000, E1   -75.175, E3 +8303.499}
SPL {X  -154.068, Y  +736.353, Z    +0.000, E1   -74.906, E3 +8310.674}
SPL {X  -149.738, Y  +746.340, Z    +0.000, E1   -74.451, E3 +8320.361}
SPL {X  -144.163, Y  +757.090, Z    +0.000, E1   -74.033, E3 +8329.454}
SPL {X  -139.284, Y  +765.165, Z    +0.000, E1   -73.322, E3 +8339.149}
SPL {X  -134.662, Y  +771.969, Z    +0.000, E1   -72.884, E3 +8345.480}
SPL {X  -131.459, Y  +776.289, Z    +0.000, E1   -72.475, E3 +8350.147}
SPL {X  -127.605, Y  +781.126, Z    +0.000, E1   -71.922, E3 +8355.592}
SPL {X  -124.773, Y  +784.457, Z    +0.000, E1   -71.383, E3 +8359.639}
SPL {X  -119.086, Y  +790.645, Z    +0.000, E1   -72.931, E3 +8356.493}
SPL {X   -51.449, Y  +832.958, Z    +0.000, E1   -57.230, E3 +8514.013}
ENDSPLINE

SPLINE
SPL {X  -123.821, Y  +785.537, Z    +0.000, E1   -64.536, E3 +8715.758}
SPL {X  -153.467, Y  +737.853, Z    +0.000, E1   -51.757, E3 +8718.073}
SPL {X  -161.000, Y  +714.475, Z    +0.000, E1   -39.424, E3 +8717.546}
SPL {X  -164.534, Y  +694.695, Z    +0.000, E1   -23.511, E3 +8715.835}
SPL {X  -165.597, Y  +679.703, Z    +0.000, E1    -7.645, E3 +8715.711}
SPL {X  -165.650, Y  +673.520, Z    +0.000, E1    -0.048, E3 +8714.663}
SPL {X  -165.650, Y  +671.692, Z    +0.000, E1    +4.450, E3 +8714.230}
SPL {X  -165.650, Y  +667.743, Z    +0.000, E1   +15.617, E3 +8714.147}
SPL {X  -165.650, Y  +662.891, Z    +0.000, E1   +29.740, E3 +8713.665}
SPL {X  -165.650, Y  +658.373, Z    +0.000, E1   +40.877, E3 +8713.863}
SPL {X  -165.650, Y  +650.834, Z    +0.000, E1   +55.143, E3 +8713.116}
SPL {X  -165.650, Y  +639.785, Z    +0.000, E1   +67.512, E3 +8712.333}
SPL {X  -165.650, Y  +619.979, Z    +0.000, E1   +79.465, E3 +8708.502}
SPL {X  -165.650, Y  +584.722, Z    +0.000, E1   +79.551, E3 +8717.793}
SPL {X  -165.650, Y  +560.326, Z    +0.000, E1   +78.360, E3 +8727.515}
SPL {X  -160.258, Y  +336.579, Z    +0.000, E1   +78.314, E3 +8799.037}
SPL {X  -159.618, Y  +334.207, Z    +0.000, E1   +75.622, E3 +8829.851}
SPL {X  -156.487, Y  +324.170, Z    +0.000, E1   +75.150, E3 +8840.207}
SPL {X  -142.256, Y  +293.629, Z    +0.000, E1   +77.020, E3 +8835.306}
ENDSPLINE

SPLINE
SPL {X  -142.811, Y  +294.566, Z    +0.000, E1   +75.668, E3 +8847.269}
ENDSPLINE

SPLINE
SPL {X  -141.646, Y  +292.615, Z    +0.000, E1   +74.702, E3 +8856.362}
SPL {X  -140.419, Y  +290.622, Z    +0.000, E1   +73.705, E3 +8865.205}
SPL {X  -136.008, Y  +283.940, Z    +0.000, E1   +73.594, E3 +8869.325}
SPL {X  -132.748, Y  +279.415, Z    +0.000, E1   +73.006, E3 +8875.380}
SPL {X  -129.007, Y  +274.590, Z    +0.000, E1   +72.484, E3 +8880.729}
SPL {X  -125.914, Y  +270.864, Z    +0.000, E1   +72.144, E3 +8884.221}
SPL {X  -123.729, Y  +268.359, Z    +0.000, E1   +71.932, E3 +8886.393}
SPL {X  -111.023, Y  +255.562, Z    +0.000, E1   +75.772, E3 +8877.259}
SPL {X   -52.752, Y  +221.474, Z    +0.000, E1   +59.157, E3 +9006.511}
SPL {X   -49.901, Y  +220.545, Z    +0.000, E1   +56.696, E3 +9092.903}
ENDSPLINE

SPLINE
SPL {X  -127.117, Y  +272.287, Z    +0.000, E1   +62.713, E3 +9239.196}
SPL {X  -154.956, Y  +319.945, Z    +0.000, E1   +49.402, E3 +9243.595}
SPL {X  -162.871, Y  +348.286, Z    +0.000, E1   +32.462, E3 +9242.623}
SPL {X  -165.127, Y  +365.342, Z    +0.000, E1   +17.250, E3 +9242.461}
SPL {X  -165.640, Y  +376.693, Z    +0.000, E1    +4.721, E3 +9242.034}
SPL {X  -165.650, Y  +380.500, Z    +0.000, E1    -0.000, E3 +9241.185}
SPL {X  -165.650, Y  +383.262, Z    +0.000, E1    -6.645, E3 +9240.714}
SPL {X  -165.650, Y  +388.390, Z    +0.000, E1   -21.508, E3 +9240.502}
SPL {X  -165.650, Y  +393.439, Z    +0.000, E1   -35.398, E3 +9240.069}
SPL {X  -165.650, Y  +400.610, Z    +0.000, E1   -50.510, E3 +9239.807}
SPL {X  -165.650, Y  +414.376, Z    +0.000, E1   -68.098, E3 +9237.841}
SPL {X  -165.650, Y  +468.582, Z    +0.000, E1   -78.237, E3 +9246.611}
SPL {X  -158.306, Y  +724.277, Z    +0.000, E1   -77.461, E3 +9337.052}
ENDSPLINE

SPLINE
SPL {X  -160.145, Y  +717.851, Z    +0.000, E1   -75.386, E3 +9357.565}
ENDSPLINE

SPLINE
SPL {X  -157.156, Y  +727.862, Z    +0.000, E1   -75.175, E3 +9365.038}
SPL {X  -154.068, Y  +736.353, Z    +0.000, E1   -74.906, E3 +9372.212}
SPL {X  -149.738, Y  +746.340, Z    +0.000, E1   -74.451, E3 +9381.900}
SPL {X  -144.163, Y  +757.090, Z    +0.000, E1   -74.033, E3 +9390.992}
SPL {X  -139.284, Y  +765.165, Z    +0.000, E1   -73.322, E3 +9400.687}
SPL {X  -134.662, Y  +771.969, Z    +0.000, E1   -72.884, E3 +9407.019}
SPL {X  -131.459, Y  +776.289, Z    +0.000, E1   -72.475, E3 +9411.686}
SPL {X  -127.605, Y  +781.126, Z    +0.000, E1   -71.922, E3 +9417.130}
SPL {X  -124.773, Y  +784.457, Z    +0.000, E1   -71.383, E3 +9421.177}
SPL {X  -119.086, Y  +790.645, Z    +0.000, E1   -72.931, E3 +9418.032}
SPL {X   -51.449, Y  +832.958, Z    +0.000, E1   -57.230, E3 +9575.551}
ENDSPLINE

SPLINE
SPL {X  -123.821, Y  +785.537, Z    +0.000, E1   -64.536, E3 +9777.297}
SPL {X  -153.467, Y  +737.853, Z    +0.000, E1   -51.757, E3 +9779.611}
SPL {X  -161.000, Y  +714.475, Z    +0.000, E1   -39.424, E3 +9779.084}
SPL {X  -164.534, Y  +694.695, Z    +0.000, E1   -23.511, E3 +9777.374}
SPL {X  -165.597, Y  +679.703, Z    +0.000, E1    -7.645, E3 +9777.250}
SPL {X  -165.650, Y  +673.520, Z    +0.000, E1    -0.048, E3 +9776.201}
SPL {X  -165.650, Y  +671.692, Z    +0.000, E1    +4.450, E3 +9775.768}
SPL {X  -165.650, Y  +667.743, Z    +0.000, E1   +15.617, E3 +9775.686}
SPL {X  -165.650, Y  +661.459, Z    +0.000, E1   +33.218, E3 +9775.266}
SPL {X  -165.650, Y  +653.296, Z    +0.000, E1   +51.333, E3 +9774.822}
SPL {X  -165.650, Y  +642.000, Z    +0.000, E1   +65.561, E3 +9774.034}
SPL {X  -165.650, Y  +619.979, Z    +0.000, E1   +79.465, E3 +9770.040}
SPL {X  -165.650, Y  +569.632, Z    +0.000, E1   +78.783, E3 +9785.319}
SPL {X  -158.840, Y  +331.491, Z    +0.000, E1   +77.462, E3 +9871.629}
ENDSPLINE

SPLINE
SPL {X  -159.893, Y  +335.208, Z    +0.000, E1   +75.483, E3 +9892.364}
ENDSPLINE

SPLINE
SPL {X  -156.487, Y  +324.170, Z    +0.000, E1   +75.150, E3 +9901.745}
SPL {X  -142.256, Y  +293.629, Z    +0.000, E1   +77.020, E3 +9896.845}
ENDSPLINE

SPLINE
SPL {X  -142.811, Y  +294.566, Z    +0.000, E1   +75.668, E3 +9908.807}
ENDSPLINE

SPLINE
SPL {X  -141.646, Y  +292.615, Z    +0.000, E1   +74.702, E3 +9917.901}
SPL {X  -140.419, Y  +290.622, Z    +0.000, E1   +73.705, E3 +9926.744}
SPL {X  -136.008, Y  +283.940, Z    +0.000, E1   +73.594, E3 +9930.863}
SPL {X  -132.748, Y  +279.415, Z    +0.000, E1   +73.006, E3 +9936.919}
SPL {X  -129.007, Y  +274.590, Z    +0.000, E1   +72.484, E3 +9942.268}
SPL {X  -125.914, Y  +270.864, Z    +0.000, E1   +72.144, E3 +9945.759}
SPL {X  -123.729, Y  +268.359, Z    +0.000, E1   +71.932, E3 +9947.932}
SPL {X  -111.023, Y  +255.562, Z    +0.000, E1   +75.772, E3 +9938.797}
SPL {X   -49.289, Y  +220.353, Z    +0.000, E1   +56.690, E3 +10131.512}
ENDSPLINE

SPLINE
SPL {X  -127.117, Y  +272.287, Z    +0.000, E1   +62.713, E3 +10300.734}
SPL {X  -154.956, Y  +319.945, Z    +0.000, E1   +49.402, E3 +10305.133}
SPL {X  -162.871, Y  +348.286, Z    +0.000, E1   +32.462, E3 +10304.161}
SPL {X  -165.127, Y  +365.342, Z    +0.000, E1   +17.250, E3 +10304.000}
SPL {X  -165.640, Y  +376.693, Z    +0.000, E1    +4.721, E3 +10303.572}
SPL {X  -165.650, Y  +380.500, Z    +0.000, E1    -0.000, E3 +10302.723}
SPL {X  -165.650, Y  +383.262, Z    +0.000, E1    -6.645, E3 +10302.253}
SPL {X  -165.650, Y  +388.390, Z    +0.000, E1   -21.508, E3 +10302.040}
SPL {X  -165.650, Y  +393.439, Z    +0.000, E1   -35.398, E3 +10301.608}
SPL {X  -165.650, Y  +400.610, Z    +0.000, E1   -50.510, E3 +10301.345}
SPL {X  -165.650, Y  +414.376, Z    +0.000, E1   -68.098, E3 +10299.379}
SPL {X  -165.650, Y  +468.582, Z    +0.000, E1   -78.237, E3 +10308.149}
SPL {X  -158.306, Y  +724.277, Z    +0.000, E1   -77.461, E3 +10398.591}
ENDSPLINE

SPLINE
SPL {X  -160.145, Y  +717.851, Z    +0.000, E1   -75.386, E3 +10419.104}
ENDSPLINE

SPLINE
SPL {X  -157.156, Y  +727.862, Z    +0.000, E1   -75.175, E3 +10426.576}
SPL {X  -154.068, Y  +736.353, Z    +0.000, E1   -74.906, E3 +10433.751}
SPL {X  -149.738, Y  +746.340, Z    +0.000, E1   -74.451, E3 +10443.438}
SPL {X  -145.204, Y  +755.223, Z    +0.000, E1   -74.188, E3 +10450.165}
SPL {X  -142.724, Y  +759.583, Z    +0.000, E1   -73.634, E3 +10456.985}
SPL {X  -138.277, Y  +766.711, Z    +0.000, E1   -73.303, E3 +10463.115}
SPL {X  -134.662, Y  +771.969, Z    +0.000, E1   -72.884, E3 +10468.557}
SPL {X  -131.459, Y  +776.289, Z    +0.000, E1   -72.475, E3 +10473.224}
SPL {X  -128.771, Y  +779.702, Z    +0.000, E1   -71.875, E3 +10478.171}
SPL {X  -125.267, Y  +783.889, Z    +0.000, E1   -71.674, E3 +10481.283}
SPL {X  -119.086, Y  +790.645, Z    +0.000, E1   -72.931, E3 +10479.570}
SPL {X   -51.449, Y  +832.958, Z    +0.000, E1   -57.230, E3 +10637.090}
ENDSPLINE

SPLINE
SPL {X  -123.821, Y  +785.537, Z    +0.000, E1   -64.536, E3 +10838.835}
SPL {X  -153.467, Y  +737.853, Z    +0.000, E1   -51.757, E3 +10841.150}
SPL {X  -162.176, Y  +709.248, Z    +0.000, E1   -35.773, E3 +10840.175}
SPL {X  -164.888, Y  +691.368, Z    +0.000, E1   -20.174, E3 +10838.613}
SPL {X  -165.597, Y  +679.703, Z    +0.000, E1    -7.645, E3 +10838.788}
SPL {X  -165.650, Y  +673.520, Z    +0.000, E1    -0.048, E3 +10837.740}
SPL {X  -165.650, Y  +671.692, Z    +0.000, E1    +4.450, E3 +10837.306}
SPL {X  -165.650, Y  +667.743, Z    +0.000, E1   +15.617, E3 +10837.224}
SPL {X  -165.650, Y  +662.891, Z    +0.000, E1   +29.740, E3 +10836.742}
SPL {X  -165.650, Y  +655.319, Z    +0.000, E1   +47.265, E3 +10836.591}
SPL {X  -165.650, Y  +642.000, Z    +0.000, E1   +65.561, E3 +10835.572}
SPL {X  -165.650, Y  +619.979, Z    +0.000, E1   +79.465, E3 +10831.579}
SPL {X  -165.650, Y  +569.632, Z    +0.000, E1   +78.783, E3 +10846.858}
SPL {X  -160.258, Y  +336.579, Z    +0.000, E1   +78.314, E3 +10922.114}
SPL {X  -159.618, Y  +334.207, Z    +0.000, E1   +75.622, E3 +10952.928}
SPL {X  -156.487, Y  +324.170, Z    +0.000, E1   +75.150, E3 +10963.283}
SPL {X  -142.256, Y  +293.629, Z    +0.000, E1   +77.020, E3 +10958.383}
ENDSPLINE

SPLINE
SPL {X  -142.811, Y  +294.566, Z    +0.000, E1   +75.668, E3 +10970.346}
ENDSPLINE

SPLINE
SPL {X  -141.646, Y  +292.615, Z    +0.000, E1   +74.702, E3 +10979.439}
SPL {X  -140.419, Y  +290.622, Z    +0.000, E1   +73.705, E3 +10988.282}
SPL {X  -136.008, Y  +283.940, Z    +0.000, E1   +73.594, E3 +10992.401}
SPL {X  -132.748, Y  +279.415, Z    +0.000, E1   +73.006, E3 +10998.457}
SPL {X  -129.007, Y  +274.590, Z    +0.000, E1   +72.484, E3 +11003.806}
SPL {X  -125.914, Y  +270.864, Z    +0.000, E1   +72.144, E3 +11007.298}
SPL {X  -123.729, Y  +268.359, Z    +0.000, E1   +71.932, E3 +11009.470}
SPL {X  -111.023, Y  +255.562, Z    +0.000, E1   +75.772, E3 +11000.336}
SPL {X   -49.289, Y  +220.353, Z    +0.000, E1   +56.690, E3 +11193.051}
ENDSPLINE

SPLINE
SPL {X  -127.117, Y  +272.287, Z    +0.000, E1   +62.713, E3 +11362.273}
SPL {X  -152.442, Y  +313.682, Z    +0.000, E1   +51.943, E3 +11366.505}
SPL {X  -159.925, Y  +335.326, Z    +0.000, E1   +41.361, E3 +11366.447}
SPL {X  -163.450, Y  +351.595, Z    +0.000, E1   +29.785, E3 +11365.558}
SPL {X  -165.127, Y  +365.342, Z    +0.000, E1   +17.250, E3 +11365.538}
SPL {X  -165.640, Y  +376.693, Z    +0.000, E1    +4.721, E3 +11365.111}
SPL {X  -165.650, Y  +380.500, Z    +0.000, E1    -0.000, E3 +11364.262}
SPL {X  -165.650, Y  +382.123, Z    +0.000, E1    -3.912, E3 +11363.889}
SPL {X  -165.650, Y  +387.069, Z    +0.000, E1   -17.420, E3 +11363.600}
SPL {X  -165.650, Y  +393.439, Z    +0.000, E1   -35.398, E3 +11363.146}
SPL {X  -165.650, Y  +400.610, Z    +0.000, E1   -50.510, E3 +11362.884}
SPL {X  -165.650, Y  +414.376, Z    +0.000, E1   -68.098, E3 +11360.917}
SPL {X  -165.650, Y  +468.582, Z    +0.000, E1   -78.237, E3 +11369.688}
SPL {X  -160.244, Y  +717.475, Z    +0.000, E1   -78.917, E3 +11442.246}
SPL {X  -159.651, Y  +719.676, Z    +0.000, E1   -75.661, E3 +11478.632}
SPL {X  -157.156, Y  +727.862, Z    +0.000, E1   -75.175, E3 +11488.114}
SPL {X  -152.814, Y  +739.436, Z    +0.000, E1   -74.813, E3 +11497.968}
SPL {X  -148.754, Y  +748.385, Z    +0.000, E1   -74.281, E3 +11507.410}
SPL {X  -144.163, Y  +757.090, Z    +0.000, E1   -74.033, E3 +11514.069}
SPL {X  -139.284, Y  +765.165, Z    +0.000, E1   -73.322, E3 +11523.764}
SPL {X  -134.662, Y  +771.969, Z    +0.000, E1   -72.884, E3 +11530.096}
SPL {X  -131.459, Y  +776.289, Z    +0.000, E1   -72.475, E3 +11534.763}
SPL {X  -128.771, Y  +779.702, Z    +0.000, E1   -71.875, E3 +11539.709}
SPL {X  -124.506, Y  +784.762, Z    +0.000, E1   -71.815, E3 +11542.598}
SPL {X  -112.958, Y  +796.663, Z    +0.000, E1   -74.119, E3 +11539.301}
SPL {X   -54.274, Y  +832.006, Z    +0.000, E1   -58.502, E3 +11671.321}
SPL {X   -50.797, Y  +833.169, Z    +0.000, E1   -57.000, E3 +11766.670}
ENDSPLINE

SPLINE
SPL {X  -113.713, Y  +795.955, Z    +0.000, E1   -65.735, E3 +11897.547}
SPL {X  -131.116, Y  +776.736, Z    +0.000, E1   -63.149, E3 +11902.077}
SPL {X  -153.467, Y  +737.853, Z    +0.000, E1   -51.757, E3 +11902.688}
SPL {X  -162.176, Y  +709.248, Z    +0.000, E1   -35.773, E3 +11901.714}
SPL {X  -164.888, Y  +691.368, Z    +0.000, E1   -20.174, E3 +11900.151}
SPL {X  -165.597, Y  +679.703, Z    +0.000, E1    -7.645, E3 +11900.327}
SPL {X  -165.650, Y  +673.520, Z    +0.000, E1    -0.048, E3 +11899.278}
SPL {X  -165.650, Y  +671.692, Z    +0.000, E1    +4.450, E3 +11898.845}
SPL {X  -165.650, Y  +667.743, Z    +0.000, E1   +15.617, E3 +11898.763}
SPL {X  -165.650, Y  +662.891, Z    +0.000, E1   +29.740, E3 +11898.281}
SPL {X  -165.650, Y  +655.319, Z    +0.000, E1   +47.265, E3 +11898.129}
SPL {X  -165.650, Y  +642.000, Z    +0.000, E1   +65.561, E3 +11897.111}
SPL {X  -165.650, Y  +619.979, Z    +0.000, E1   +79.465, E3 +11893.117}
SPL {X  -165.650, Y  +569.632, Z    +0.000, E1   +78.783, E3 +11908.396}
SPL {X  -158.840, Y  +331.491, Z    +0.000, E1   +77.462, E3 +11994.706}
ENDSPLINE

SPLINE
SPL {X  -159.893, Y  +335.208, Z    +0.000, E1   +75.483, E3 +12015.441}
ENDSPLINE

SPLINE
SPL {X  -156.487, Y  +324.170, Z    +0.000, E1   +75.150, E3 +12024.822}
SPL {X  -142.256, Y  +293.629, Z    +0.000, E1   +77.020, E3 +12019.922}
ENDSPLINE

SPLINE
SPL {X  -142.811, Y  +294.566, Z    +0.000, E1   +75.668, E3 +12031.884}
ENDSPLINE

SPLINE
SPL {X  -141.646, Y  +292.615, Z    +0.000, E1   +74.702, E3 +12040.978}
SPL {X  -140.419, Y  +290.622, Z    +0.000, E1   +73.705, E3 +12049.821}
SPL {X  -135.839, Y  +283.697, Z    +0.000, E1   +73.388, E3 +12055.559}
SPL {X  -131.336, Y  +277.551, Z    +0.000, E1   +72.879, E3 +12061.811}
SPL {X  -126.848, Y  +271.966, Z    +0.000, E1   +72.322, E3 +12067.540}
SPL {X  -123.729, Y  +268.359, Z    +0.000, E1   +71.932, E3 +12071.008}
SPL {X  -111.023, Y  +255.562, Z    +0.000, E1   +75.772, E3 +12061.874}
SPL {X   -52.752, Y  +221.474, Z    +0.000, E1   +59.157, E3 +12191.126}
SPL {X   -49.901, Y  +220.545, Z    +0.000, E1   +56.696, E3 +12277.518}
ENDSPLINE

SPLINE
SPL {X  -127.117, Y  +272.287, Z    +0.000, E1   +62.713, E3 +12423.811}
SPL {X  -152.442, Y  +313.682, Z    +0.000, E1   +51.943, E3 +12428.043}
SPL {X  -162.319, Y  +345.447, Z    +0.000, E1   +34.671, E3 +12427.468}
SPL {X  -165.127, Y  +365.342, Z    +0.000, E1   +17.250, E3 +12427.076}
SPL {X  -165.640, Y  +376.693, Z    +0.000, E1    +4.721, E3 +12426.649}
SPL {X  -165.650, Y  +380.500, Z    +0.000, E1    -0.000, E3 +12425.800}
SPL {X  -165.650, Y  +383.262, Z    +0.000, E1    -6.645, E3 +12425.329}
SPL {X  -165.650, Y  +388.390, Z    +0.000, E1   -21.508, E3 +12425.117}
SPL {X  -165.650, Y  +393.439, Z    +0.000, E1   -35.398, E3 +12424.685}
SPL {X  -165.650, Y  +400.610, Z    +0.000, E1   -50.510, E3 +12424.422}
SPL {X  -165.650, Y  +414.376, Z    +0.000, E1   -68.098, E3 +12422.456}
SPL {X  -165.650, Y  +468.582, Z    +0.000, E1   -78.237, E3 +12431.226}
SPL {X  -158.306, Y  +724.277, Z    +0.000, E1   -77.461, E3 +12521.667}
ENDSPLINE

SPLINE
SPL {X  -160.145, Y  +717.851, Z    +0.000, E1   -75.386, E3 +12542.181}
ENDSPLINE

SPLINE
SPL {X  -157.156, Y  +727.862, Z    +0.000, E1   -75.175, E3 +12549.653}
SPL {X  -152.814, Y  +739.436, Z    +0.000, E1   -74.813, E3 +12559.507}
SPL {X  -148.754, Y  +748.385, Z    +0.000, E1   -74.281, E3 +12568.949}
SPL {X  -144.163, Y  +757.090, Z    +0.000, E1   -74.033, E3 +12575.608}
SPL {X  -139.284, Y  +765.165, Z    +0.000, E1   -73.322, E3 +12585.302}
SPL {X  -134.662, Y  +771.969, Z    +0.000, E1   -72.884, E3 +12591.634}
SPL {X  -131.459, Y  +776.289, Z    +0.000, E1   -72.475, E3 +12596.301}
SPL {X  -127.605, Y  +781.126, Z    +0.000, E1   -71.922, E3 +12601.745}
SPL {X  -124.773, Y  +784.457, Z    +0.000, E1   -71.383, E3 +12605.793}
SPL {X  -119.086, Y  +790.645, Z    +0.000, E1   -72.931, E3 +12602.647}
SPL {X   -51.449, Y  +832.958, Z    +0.000, E1   -57.230, E3 +12760.167}
ENDSPLINE

SPLINE
SPL {X  -123.821, Y  +785.537, Z    +0.000, E1   -64.536, E3 +12961.912}
SPL {X  -153.467, Y  +737.853, Z    +0.000, E1   -51.757, E3 +12964.227}
SPL {X  -162.176, Y  +709.248, Z    +0.000, E1   -35.773, E3 +12963.252}
SPL {X  -164.888, Y  +691.368, Z    +0.000, E1   -20.174, E3 +12961.690}
SPL {X  -165.597, Y  +679.703, Z    +0.000, E1    -7.645, E3 +12961.865}
SPL {X  -165.650, Y  +673.520, Z    +0.000, E1    -0.048, E3 +12960.817}
SPL {X  -165.650, Y  +671.692, Z    +0.000, E1    +4.450, E3 +12960.383}
SPL {X  -165.650, Y  +667.743, Z    +0.000, E1   +15.617, E3 +12960.301}
SPL {X  -165.650, Y  +661.459, Z    +0.000, E1   +33.218, E3 +12959.882}
SPL {X  -165.650, Y  +653.296, Z    +0.000, E1   +51.333, E3 +12959.437}
SPL {X  -165.650, Y  +642.000, Z    +0.000, E1   +65.561, E3 +12958.649}
SPL {X  -165.650, Y  +619.979, Z    +0.000, E1   +79.465, E3 +12954.656}
SPL {X  -165.650, Y  +584.722, Z    +0.000, E1   +79.551, E3 +12963.947}
SPL {X  -165.650, Y  +560.326, Z    +0.000, E1   +78.360, E3 +12973.669}
SPL {X  -158.840, Y  +331.491, Z    +0.000, E1   +77.462, E3 +13056.245}
ENDSPLINE

SPLINE
SPL {X  -159.893, Y  +335.208, Z    +0.000, E1   +75.483, E3 +13076.979}
ENDSPLINE

SPLINE
SPL {X  -156.487, Y  +324.170, Z    +0.000, E1   +75.150, E3 +13086.360}
SPL {X  -142.256, Y  +293.629, Z    +0.000, E1   +77.020, E3 +13081.460}
ENDSPLINE

SPLINE
SPL {X  -142.811, Y  +294.566, Z    +0.000, E1   +75.668, E3 +13093.422}
ENDSPLINE

SPLINE
SPL {X  -141.646, Y  +292.615, Z    +0.000, E1   +74.702, E3 +13102.516}
SPL {X  -140.419, Y  +290.622, Z    +0.000, E1   +73.705, E3 +13111.359}
SPL {X  -136.008, Y  +283.940, Z    +0.000, E1   +73.594, E3 +13115.478}
SPL {X  -132.748, Y  +279.415, Z    +0.000, E1   +73.006, E3 +13121.534}
SPL {X  -129.007, Y  +274.590, Z    +0.000, E1   +72.484, E3 +13126.883}
SPL {X  -124.646, Y  +269.397, Z    +0.000, E1   +72.041, E3 +13131.631}
SPL {X  -111.023, Y  +255.562, Z    +0.000, E1   +75.772, E3 +13123.413}
SPL {X   -52.752, Y  +221.474, Z    +0.000, E1   +59.157, E3 +13252.664}
SPL {X   -49.901, Y  +220.545, Z    +0.000, E1   +56.696, E3 +13339.057}
ENDSPLINE

SPLINE
SPL {X  -127.117, Y  +272.287, Z    +0.000, E1   +62.713, E3 +13485.350}
SPL {X  -152.442, Y  +313.682, Z    +0.000, E1   +51.943, E3 +13489.581}
SPL {X  -159.925, Y  +335.326, Z    +0.000, E1   +41.361, E3 +13489.523}
SPL {X  -163.450, Y  +351.595, Z    +0.000, E1   +29.785, E3 +13488.635}
SPL {X  -165.127, Y  +365.342, Z    +0.000, E1   +17.250, E3 +13488.615}
SPL {X  -165.640, Y  +376.693, Z    +0.000, E1    +4.721, E3 +13488.188}
SPL {X  -165.650, Y  +380.500, Z    +0.000, E1    -0.000, E3 +13487.339}
SPL {X  -165.650, Y  +383.262, Z    +0.000, E1    -6.645, E3 +13486.868}
SPL {X  -165.650, Y  +388.390, Z    +0.000, E1   -21.508, E3 +13486.656}
SPL {X  -165.650, Y  +393.439, Z    +0.000, E1   -35.398, E3 +13486.223}
SPL {X  -165.650, Y  +400.610, Z    +0.000, E1   -50.510, E3 +13485.961}
SPL {X  -165.650, Y  +414.376, Z    +0.000, E1   -68.098, E3 +13483.994}
SPL {X  -165.650, Y  +468.582, Z    +0.000, E1   -78.237, E3 +13492.765}
SPL {X  -158.306, Y  +724.277, Z    +0.000, E1   -77.461, E3 +13583.206}
ENDSPLINE

SPLINE
SPL {X  -160.145, Y  +717.851, Z    +0.000, E1   -75.386, E3 +13603.719}
ENDSPLINE

SPLINE
SPL {X  -157.156, Y  +727.862, Z    +0.000, E1   -75.175, E3 +13611.191}
SPL {X  -152.814, Y  +739.436, Z    +0.000, E1   -74.813, E3 +13621.045}
SPL {X  -147.104, Y  +751.659, Z    +0.000, E1   -74.255, E3 +13632.490}
SPL {X  -142.724, Y  +759.583, Z    +0.000, E1   -73.634, E3 +13641.600}
SPL {X  -138.277, Y  +766.711, Z    +0.000, E1   -73.303, E3 +13647.730}
SPL {X  -134.662, Y  +771.969, Z    +0.000, E1   -72.884, E3 +13653.173}
SPL {X  -131.459, Y  +776.289, Z    +0.000, E1   -72.475, E3 +13657.840}
SPL {X  -128.771, Y  +779.702, Z    +0.000, E1   -71.875, E3 +13662.786}
SPL {X  -125.267, Y  +783.889, Z    +0.000, E1   -71.674, E3 +13665.899}
SPL {X  -119.086, Y  +790.645, Z    +0.000, E1   -72.931, E3 +13664.185}
SPL {X   -51.449, Y  +832.958, Z    +0.000, E1   -57.230, E3 +13821.705}
ENDSPLINE

SPLINE
SPL {X  -123.821, Y  +785.537, Z    +0.000, E1   -64.536, E3 +14023.450}
SPL {X  -153.467, Y  +737.853, Z    +0.000, E1   -51.757, E3 +14025.765}
SPL {X  -162.176, Y  +709.248, Z    +0.000, E1   -35.773, E3 +14024.791}
SPL {X  -164.888, Y  +691.368, Z    +0.000, E1   -20.174, E3 +14023.228}
SPL {X  -165.597, Y  +679.703, Z    +0.000, E1    -7.645, E3 +14023.403}
SPL {X  -165.650, Y  +673.520, Z    +0.000, E1    -0.048, E3 +14022.355}
SPL {X  -165.650, Y  +671.692, Z    +0.000, E1    +4.450, E3 +14021.922}
SPL {X  -165.650, Y  +667.743, Z    +0.000, E1   +15.617, E3 +14021.840}
SPL {X  -165.650, Y  +662.891, Z    +0.000, E1   +29.740, E3 +14021.358}
SPL {X  -165.650, Y  +655.319, Z    +0.000, E1   +47.265, E3 +14021.206}
SPL {X  -165.650, Y  +642.000, Z    +0.000, E1   +65.561, E3 +14020.188}
SPL {X  -165.650, Y  +619.979, Z    +0.000, E1   +79.465, E3 +14016.194}
SPL {X  -165.650, Y  +569.632, Z    +0.000, E1   +78.783, E3 +14031.473}
SPL {X  -160.258, Y  +336.579, Z    +0.000, E1   +78.314, E3 +14106.729}
SPL {X  -159.618, Y  +334.207, Z    +0.000, E1   +75.622, E3 +14137.543}
SPL {X  -156.487, Y  +324.170, Z    +0.000, E1   +75.150, E3 +14147.899}
SPL {X  -142.256, Y  +293.629, Z    +0.000, E1   +77.020, E3 +14142.999}
ENDSPLINE

SPLINE
SPL {X  -142.811, Y  +294.566, Z    +0.000, E1   +75.668, E3 +14154.961}
ENDSPLINE

SPLINE
SPL {X  -141.646, Y  +292.615, Z    +0.000, E1   +74.702, E3 +14164.055}
SPL {X  -140.419, Y  +290.622, Z    +0.000, E1   +73.705, E3 +14172.898}
SPL {X  -136.008, Y  +283.940, Z    +0.000, E1   +73.594, E3 +14177.017}
SPL {X  -132.748, Y  +279.415, Z    +0.000, E1   +73.006, E3 +14183.073}
SPL {X  -129.007, Y  +274.590, Z    +0.000, E1   +72.484, E3 +14188.421}
SPL {X  -125.914, Y  +270.864, Z    +0.000, E1   +72.144, E3 +14191.913}
SPL {X  -123.729, Y  +268.359, Z    +0.000, E1   +71.932, E3 +14194.085}
SPL {X  -111.023, Y  +255.562, Z    +0.000, E1   +75.772, E3 +14184.951}
SPL {X   -52.752, Y  +221.474, Z    +0.000, E1   +59.157, E3 +14314.203}
SPL {X   -49.901, Y  +220.545, Z    +0.000, E1   +56.696, E3 +14400.595}
ENDSPLINE

SPLINE
SPL {X  -127.117, Y  +272.287, Z    +0.000, E1   +62.713, E3 +14546.888}
SPL {X  -152.442, Y  +313.682, Z    +0.000, E1   +51.943, E3 +14551.120}
SPL {X  -162.319, Y  +345.447, Z    +0.000, E1   +34.671, E3 +14550.545}
SPL {X  -165.127, Y  +365.342, Z    +0.000, E1   +17.250, E3 +14550.153}
SPL {X  -165.640, Y  +376.693, Z    +0.000, E1    +4.721, E3 +14549.726}
SPL {X  -165.650, Y  +380.500, Z    +0.000, E1    -0.000, E3 +14548.877}
SPL {X  -165.650, Y  +382.123, Z    +0.000, E1    -3.912, E3 +14548.504}
SPL {X  -165.650, Y  +387.069, Z    +0.000, E1   -17.420, E3 +14548.216}
SPL {X  -165.650, Y  +393.439, Z    +0.000, E1   -35.398, E3 +14547.762}
SPL {X  -165.650, Y  +400.610, Z    +0.000, E1   -50.510, E3 +14547.499}
SPL {X  -165.650, Y  +414.376, Z    +0.000, E1   -68.098, E3 +14545.533}
SPL {X  -165.650, Y  +468.582, Z    +0.000, E1   -78.237, E3 +14554.303}
SPL {X  -160.244, Y  +717.475, Z    +0.000, E1   -78.917, E3 +14626.861}
SPL {X  -159.651, Y  +719.676, Z    +0.000, E1   -75.661, E3 +14663.248}
SPL {X  -157.156, Y  +727.862, Z    +0.000, E1   -75.175, E3 +14672.730}
SPL {X  -154.068, Y  +736.353, Z    +0.000, E1   -74.906, E3 +14679.905}
SPL {X  -149.738, Y  +746.340, Z    +0.000, E1   -74.451, E3 +14689.592}
SPL {X  -144.163, Y  +757.090, Z    +0.000, E1   -74.033, E3 +14698.685}
SPL {X  -139.284, Y  +765.165, Z    +0.000, E1   -73.322, E3 +14708.379}
SPL {X  -134.662, Y  +771.969, Z    +0.000, E1   -72.884, E3 +14714.711}
SPL {X  -131.459, Y  +776.289, Z    +0.000, E1   -72.475, E3 +14719.378}
SPL {X  -127.605, Y  +781.126, Z    +0.000, E1   -71.922, E3 +14724.822}
SPL {X  -124.773, Y  +784.457, Z    +0.000, E1   -71.383, E3 +14728.870}
SPL {X  -119.086, Y  +790.645, Z    +0.000, E1   -72.931, E3 +14725.724}
SPL {X   -51.449, Y  +832.958, Z    +0.000, E1   -57.230, E3 +14883.244}
ENDSPLINE

SPLINE
SPL {X  -123.821, Y  +785.537, Z    +0.000, E1   -64.536, E3 +15084.989}
SPL {X  -153.467, Y  +737.853, Z    +0.000, E1   -51.757, E3 +15087.304}
SPL {X  -161.000, Y  +714.475, Z    +0.000, E1   -39.424, E3 +15086.776}
SPL {X  -164.534, Y  +694.695, Z    +0.000, E1   -23.511, E3 +15085.066}
SPL {X  -165.597, Y  +679.703, Z    +0.000, E1    -7.645, E3 +15084.942}
SPL {X  -165.650, Y  +673.520, Z    +0.000, E1    -0.048, E3 +15083.894}
SPL {X  -165.650, Y  +671.692, Z    +0.000, E1    +4.450, E3 +15083.460}
SPL {X  -165.650, Y  +667.743, Z    +0.000, E1   +15.617, E3 +15083.378}
SPL {X  -165.650, Y  +662.891, Z    +0.000, E1   +29.740, E3 +15082.896}
SPL {X  -165.650, Y  +658.373, Z    +0.000, E1   +40.877, E3 +15083.093}
SPL {X  -165.650, Y  +650.834, Z    +0.000, E1   +55.143, E3 +15082.347}
SPL {X  -165.650, Y  +639.785, Z    +0.000, E1   +67.512, E3 +15081.564}
SPL {X  -165.650, Y  +619.979, Z    +0.000, E1   +79.465, E3 +15077.733}
SPL {X  -165.650, Y  +584.722, Z    +0.000, E1   +79.551, E3 +15087.023}
SPL {X  -165.650, Y  +560.326, Z    +0.000, E1   +78.360, E3 +15096.746}
SPL {X  -160.258, Y  +336.579, Z    +0.000, E1   +78.314, E3 +15168.268}
SPL {X  -159.618, Y  +334.207, Z    +0.000, E1   +75.622, E3 +15199.082}
SPL {X  -156.487, Y  +324.170, Z    +0.000, E1   +75.150, E3 +15209.437}
SPL {X  -142.256, Y  +293.629, Z    +0.000, E1   +77.020, E3 +15204.537}
ENDSPLINE

SPLINE
SPL {X  -142.811, Y  +294.566, Z    +0.000, E1   +75.668, E3 +15216.499}
ENDSPLINE

SPLINE
SPL {X  -141.646, Y  +292.615, Z    +0.000, E1   +74.702, E3 +15225.593}
SPL {X  -140.419, Y  +290.622, Z    +0.000, E1   +73.705, E3 +15234.436}
SPL {X  -136.008, Y  +283.940, Z    +0.000, E1   +73.594, E3 +15238.555}
SPL {X  -132.748, Y  +279.415, Z    +0.000, E1   +73.006, E3 +15244.611}
SPL {X  -129.007, Y  +274.590, Z    +0.000, E1   +72.484, E3 +15249.960}
SPL {X  -125.914, Y  +270.864, Z    +0.000, E1   +72.144, E3 +15253.451}
SPL {X  -123.729, Y  +268.359, Z    +0.000, E1   +71.932, E3 +15255.624}
SPL {X  -111.023, Y  +255.562, Z    +0.000, E1   +75.772, E3 +15246.490}
SPL {X   -49.289, Y  +220.353, Z    +0.000, E1   +56.690, E3 +15439.205}
ENDSPLINE

SPLINE
SPL {X  -127.117, Y  +272.287, Z    +0.000, E1   +62.713, E3 +15608.427}
SPL {X  -154.956, Y  +319.945, Z    +0.000, E1   +49.402, E3 +15612.826}
SPL {X  -162.871, Y  +348.286, Z    +0.000, E1   +32.462, E3 +15611.853}
SPL {X  -165.127, Y  +365.342, Z    +0.000, E1   +17.250, E3 +15611.692}
SPL {X  -165.640, Y  +376.693, Z    +0.000, E1    +4.721, E3 +15611.265}
SPL {X  -165.650, Y  +380.500, Z    +0.000, E1    -0.000, E3 +15610.416}
SPL {X  -165.650, Y  +382.123, Z    +0.000, E1    -3.912, E3 +15610.043}
SPL {X  -165.650, Y  +387.069, Z    +0.000, E1   -17.420, E3 +15609.754}
SPL {X  -165.650, Y  +393.439, Z    +0.000, E1   -35.398, E3 +15609.300}
SPL {X  -165.650, Y  +400.610, Z    +0.000, E1   -50.510, E3 +15609.038}
SPL {X  -165.650, Y  +414.376, Z    +0.000, E1   -68.098, E3 +15607.071}
SPL {X  -165.650, Y  +468.582, Z    +0.000, E1   -78.237, E3 +15615.841}
SPL {X  -160.244, Y  +717.475, Z    +0.000, E1   -78.917, E3 +15688.399}
SPL {X  -159.651, Y  +719.676, Z    +0.000, E1   -75.661, E3 +15724.786}
SPL {X  -157.156, Y  +727.862, Z    +0.000, E1   -75.175, E3 +15734.268}
SPL {X  -154.068, Y  +736.353, Z    +0.000, E1   -74.906, E3 +15741.443}
SPL {X  -149.738, Y  +746.340, Z    +0.000, E1   -74.451, E3 +15751.131}
SPL {X  -144.163, Y  +757.090, Z    +0.000, E1   -74.033, E3 +15760.223}
SPL {X  -139.284, Y  +765.165, Z    +0.000, E1   -73.322, E3 +15769.918}
SPL {X  -134.662, Y  +771.969, Z    +0.000, E1   -72.884, E3 +15776.249}
SPL {X  -131.459, Y  +776.289, Z    +0.000, E1   -72.475, E3 +15780.917}
SPL {X  -127.605, Y  +781.126, Z    +0.000, E1   -71.922, E3 +15786.361}
SPL {X  -124.773, Y  +784.457, Z    +0.000, E1   -71.383, E3 +15790.408}
SPL {X  -119.086, Y  +790.645, Z    +0.000, E1   -72.931, E3 +15787.262}
SPL {X   -51.449, Y  +832.958, Z    +0.000, E1   -57.230, E3 +15944.782}
ENDSPLINE

SPLINE
SPL {X  -123.821, Y  +785.537, Z    +0.000, E1   -64.536, E3 +16146.527}
SPL {X  -153.467, Y  +737.853, Z    +0.000, E1   -51.757, E3 +16148.842}
SPL {X  -161.000, Y  +714.475, Z    +0.000, E1   -39.424, E3 +16148.315}
SPL {X  -164.534, Y  +694.695, Z    +0.000, E1   -23.511, E3 +16146.605}
SPL {X  -165.597, Y  +679.703, Z    +0.000, E1    -7.645, E3 +16146.480}
SPL {X  -165.650, Y  +673.520, Z    +0.000, E1    -0.048, E3 +16145.432}
SPL {X  -165.650, Y  +671.692, Z    +0.000, E1    +4.450, E3 +16144.999}
SPL {X  -165.650, Y  +667.743, Z    +0.000, E1   +15.617, E3 +16144.917}
SPL {X  -165.650, Y  +661.459, Z    +0.000, E1   +33.218, E3 +16144.497}
SPL {X  -165.650, Y  +653.296, Z    +0.000, E1   +51.333, E3 +16144.052}
SPL {X  -165.650, Y  +642.000, Z    +0.000, E1   +65.561, E3 +16143.265}
SPL {X  -165.650, Y  +619.979, Z    +0.000, E1   +79.465, E3 +16139.271}
SPL {X  -165.650, Y  +569.632, Z    +0.000, E1   +78.783, E3 +16154.550}
SPL {X  -158.840, Y  +331.491, Z    +0.000, E1   +77.462, E3 +16240.860}
ENDSPLINE

SPLINE
SPL {X  -159.893, Y  +335.208, Z    +0.000, E1   +75.483, E3 +16261.595}
ENDSPLINE

SPLINE
SPL {X  -156.487, Y  +324.170, Z    +0.000, E1   +75.150, E3 +16270.976}
SPL {X  -142.256, Y  +293.629, Z    +0.000, E1   +77.020, E3 +16266.076}
ENDSPLINE

SPLINE
SPL {X  -142.811, Y  +294.566, Z    +0.000, E1   +75.668, E3 +16278.038}
ENDSPLINE

SPLINE
SPL {X  -141.646, Y  +292.615, Z    +0.000, E1   +74.702, E3 +16287.131}
SPL {X  -140.419, Y  +290.622, Z    +0.000, E1   +73.705, E3 +16295.975}
SPL {X  -136.008, Y  +283.940, Z    +0.000, E1   +73.594, E3 +16300.094}
SPL {X  -132.748, Y  +279.415, Z    +0.000, E1   +73.006, E3 +16306.150}
SPL {X  -129.007, Y  +274.590, Z    +0.000, E1   +72.484, E3 +16311.498}
SPL {X  -125.914, Y  +270.864, Z    +0.000, E1   +72.144, E3 +16314.990}
SPL {X  -123.729, Y  +268.359, Z    +0.000, E1   +71.932, E3 +16317.162}
SPL {X  -111.023, Y  +255.562, Z    +0.000, E1   +75.772, E3 +16308.028}
SPL {X   -49.289, Y  +220.353, Z    +0.000, E1   +56.690, E3 +16500.743}
ENDSPLINE

SPLINE
SPL {X  -127.117, Y  +272.287, Z    +0.000, E1   +62.713, E3 +16669.965}
SPL {X  -154.956, Y  +319.945, Z    +0.000, E1   +49.402, E3 +16674.364}
SPL {X  -162.871, Y  +348.286, Z    +0.000, E1   +32.462, E3 +16673.392}
SPL {X  -165.127, Y  +365.342, Z    +0.000, E1   +17.250, E3 +16673.230}
SPL {X  -165.640, Y  +376.693, Z    +0.000, E1    +4.721, E3 +16672.803}
SPL {X  -165.650, Y  +380.500, Z    +0.000, E1    -0.000, E3 +16671.954}
SPL {X  -165.650, Y  +383.262, Z    +0.000, E1    -6.645, E3 +16671.483}
SPL {X  -165.650, Y  +388.390, Z    +0.000, E1   -21.508, E3 +16671.271}
SPL {X  -165.650, Y  +393.439, Z    +0.000, E1   -35.398, E3 +16670.839}
SPL {X  -165.650, Y  +400.610, Z    +0.000, E1   -50.510, E3 +16670.576}
SPL {X  -165.650, Y  +414.376, Z    +0.000, E1   -68.098, E3 +16668.610}
SPL {X  -165.650, Y  +468.582, Z    +0.000, E1   -78.237, E3 +16677.380}
SPL {X  -158.306, Y  +724.277, Z    +0.000, E1   -77.461, E3 +16767.821}
ENDSPLINE

SPLINE
SPL {X  -160.145, Y  +717.851, Z    +0.000, E1   -75.386, E3 +16788.335}
ENDSPLINE

SPLINE
SPL {X  -157.156, Y  +727.862, Z    +0.000, E1   -75.175, E3 +16795.807}
SPL {X  -154.068, Y  +736.353, Z    +0.000, E1   -74.906, E3 +16802.981}
SPL {X  -149.738, Y  +746.340, Z    +0.000, E1   -74.451, E3 +16812.669}
SPL {X  -144.163, Y  +757.090, Z    +0.000, E1   -74.033, E3 +16821.762}
SPL {X  -140.473, Y  +763.291, Z    +0.000, E1   -73.478, E3 +16829.203}
SPL {X  -135.914, Y  +770.196, Z    +0.000, E1   -72.974, E3 +16836.379}
SPL {X  -131.459, Y  +776.289, Z    +0.000, E1   -72.475, E3 +16842.455}
SPL {X  -128.771, Y  +779.702, Z    +0.000, E1   -71.875, E3 +16847.402}
SPL {X  -124.506, Y  +784.762, Z    +0.000, E1   -71.815, E3 +16850.290}
SPL {X  -112.958, Y  +796.663, Z    +0.000, E1   -74.119, E3 +16846.994}
SPL {X   -51.449, Y  +832.958, Z    +0.000, E1   -57.230, E3 +17006.321}
ENDSPLINE

SPLINE
SPL {X  -123.821, Y  +785.537, Z    +0.000, E1   -64.536, E3 +17208.066}
SPL {X  -153.467, Y  +737.853, Z    +0.000, E1   -51.757, E3 +17210.381}
SPL {X  -162.176, Y  +709.248, Z    +0.000, E1   -35.773, E3 +17209.406}
SPL {X  -164.888, Y  +691.368, Z    +0.000, E1   -20.174, E3 +17207.844}
SPL {X  -165.597, Y  +679.703, Z    +0.000, E1    -7.645, E3 +17208.019}
SPL {X  -165.650, Y  +673.520, Z    +0.000, E1    -0.048, E3 +17206.971}
SPL {X  -165.650, Y  +671.692, Z    +0.000, E1    +4.450, E3 +17206.537}
SPL {X  -165.650, Y  +667.743, Z    +0.000, E1   +15.617, E3 +17206.455}
SPL {X  -165.650, Y  +661.459, Z    +0.000, E1   +33.218, E3 +17206.035}
SPL {X  -165.650, Y  +650.834, Z    +0.000, E1   +55.143, E3 +17205.423}
SPL {X  -165.650, Y  +639.785, Z    +0.000, E1   +67.512, E3 +17204.641}
SPL {X  -165.650, Y  +619.979, Z    +0.000, E1   +79.465, E3 +17200.810}
SPL {X  -165.650, Y  +569.632, Z    +0.000, E1   +78.783, E3 +17216.088}
SPL {X  -158.840, Y  +331.491, Z    +0.000, E1   +77.462, E3 +17302.398}
ENDSPLINE

SPLINE
SPL {X  -159.893, Y  +335.208, Z    +0.000, E1   +75.483, E3 +17323.133}
ENDSPLINE

SPLINE
SPL {X  -156.487, Y  +324.170, Z    +0.000, E1   +75.150, E3 +17332.514}
SPL {X  -142.256, Y  +293.629, Z    +0.000, E1   +77.020, E3 +17327.614}
ENDSPLINE

SPLINE
SPL {X  -142.811, Y  +294.566, Z    +0.000, E1   +75.668, E3 +17339.576}
ENDSPLINE

SPLINE
SPL {X  -141.646, Y  +292.615, Z    +0.000, E1   +74.702, E3 +17348.670}
SPL {X  -140.419, Y  +290.622, Z    +0.000, E1   +73.705, E3 +17357.513}
SPL {X  -136.008, Y  +283.940, Z    +0.000, E1   +73.594, E3 +17361.632}
SPL {X  -132.748, Y  +279.415, Z    +0.000, E1   +73.006, E3 +17367.688}
SPL {X  -129.007, Y  +274.590, Z    +0.000, E1   +72.484, E3 +17373.037}
SPL {X  -125.914, Y  +270.864, Z    +0.000, E1   +72.144, E3 +17376.528}
SPL {X  -123.729, Y  +268.359, Z    +0.000, E1   +71.932, E3 +17378.701}
SPL {X  -111.023, Y  +255.562, Z    +0.000, E1   +75.772, E3 +17369.567}
SPL {X   -49.289, Y  +220.353, Z    +0.000, E1   +56.690, E3 +17562.282}
ENDSPLINE

SPLINE
SPL {X  -127.117, Y  +272.287, Z    +0.000, E1   +62.713, E3 +17731.503}
SPL {X  -154.956, Y  +319.945, Z    +0.000, E1   +49.402, E3 +17735.903}
SPL {X  -162.871, Y  +348.286, Z    +0.000, E1   +32.462, E3 +17734.930}
SPL {X  -165.127, Y  +365.342, Z    +0.000, E1   +17.250, E3 +17734.769}
SPL {X  -165.640, Y  +376.693, Z    +0.000, E1    +4.721, E3 +17734.342}
SPL {X  -165.650, Y  +380.500, Z    +0.000, E1    -0.000, E3 +17733.493}
SPL {X  -165.650, Y  +383.262, Z    +0.000, E1    -6.645, E3 +17733.022}
SPL {X  -165.650, Y  +388.390, Z    +0.000, E1   -21.508, E3 +17732.809}
SPL {X  -165.650, Y  +393.439, Z    +0.000, E1   -35.398, E3 +17732.377}
SPL {X  -165.650, Y  +400.610, Z    +0.000, E1   -50.510, E3 +17732.115}
SPL {X  -165.650, Y  +414.376, Z    +0.000, E1   -68.098, E3 +17730.148}
SPL {X  -165.650, Y  +468.582, Z    +0.000, E1   -78.237, E3 +17738.918}
SPL {X  -158.306, Y  +724.277, Z    +0.000, E1   -77.461, E3 +17829.360}
ENDSPLINE

SPLINE
SPL {X  -160.145, Y  +717.851, Z    +0.000, E1   -75.386, E3 +17849.873}
ENDSPLINE

SPLINE
SPL {X  -157.156, Y  +727.862, Z    +0.000, E1   -75.175, E3 +17857.345}
SPL {X  -152.814, Y  +739.436, Z    +0.000, E1   -74.813, E3 +17867.199}
SPL {X  -147.104, Y  +751.659, Z    +0.000, E1   -74.255, E3 +17878.643}
SPL {X  -141.453, Y  +761.704, Z    +0.000, E1   -73.638, E3 +17888.856}
SPL {X  -135.914, Y  +770.196, Z    +0.000, E1   -72.974, E3 +17897.918}
SPL {X  -131.459, Y  +776.289, Z    +0.000, E1   -72.475, E3 +17903.994}
SPL {X  -127.605, Y  +781.126, Z    +0.000, E1   -71.922, E3 +17909.438}
SPL {X  -124.773, Y  +784.457, Z    +0.000, E1   -71.383, E3 +17913.485}
SPL {X  -119.086, Y  +790.645, Z    +0.000, E1   -72.931, E3 +17910.339}
SPL {X   -51.449, Y  +832.958, Z    +0.000, E1   -57.230, E3 +18067.859}
ENDSPLINE

SPLINE
SPL {X  -123.821, Y  +785.537, Z    +0.000, E1   -64.536, E3 +18269.604}
SPL {X  -153.467, Y  +737.853, Z    +0.000, E1   -51.757, E3 +18271.919}
SPL {X  -162.176, Y  +709.248, Z    +0.000, E1   -35.773, E3 +18270.945}
SPL {X  -164.888, Y  +691.368, Z    +0.000, E1   -20.174, E3 +18269.382}
SPL {X  -165.597, Y  +679.703, Z    +0.000, E1    -7.645, E3 +18269.557}
SPL {X  -165.650, Y  +673.520, Z    +0.000, E1    -0.048, E3 +18268.509}
SPL {X  -165.650, Y  +671.692, Z    +0.000, E1    +4.450, E3 +18268.076}
SPL {X  -165.650, Y  +667.743, Z    +0.000, E1   +15.617, E3 +18267.994}
SPL {X  -165.650, Y  +661.459, Z    +0.000, E1   +33.218, E3 +18267.574}
SPL {X  -165.650, Y  +653.296, Z    +0.000, E1   +51.333, E3 +18267.129}
SPL {X  -165.650, Y  +642.000, Z    +0.000, E1   +65.561, E3 +18266.341}
SPL {X  -165.650, Y  +619.979, Z    +0.000, E1   +79.465, E3 +18262.348}
SPL {X  -165.650, Y  +584.722, Z    +0.000, E1   +79.551, E3 +18271.639}
SPL {X  -165.650, Y  +560.326, Z    +0.000, E1   +78.360, E3 +18281.361}
SPL {X  -158.840, Y  +331.491, Z    +0.000, E1   +77.462, E3 +18363.937}
ENDSPLINE

SPLINE
SPL {X  -159.893, Y  +335.208, Z    +0.000, E1   +75.483, E3 +18384.672}
ENDSPLINE

SPLINE
SPL {X  -156.487, Y  +324.170, Z    +0.000, E1   +75.150, E3 +18394.053}
SPL {X  -142.256, Y  +293.629, Z    +0.000, E1   +77.020, E3 +18389.152}
ENDSPLINE

SPLINE
SPL {X  -142.811, Y  +294.566, Z    +0.000, E1   +75.668, E3 +18401.115}
ENDSPLINE

SPLINE
SPL {X  -141.646, Y  +292.615, Z    +0.000, E1   +74.702, E3 +18410.208}
SPL {X  -140.419, Y  +290.622, Z    +0.000, E1   +73.705, E3 +18419.052}
SPL {X  -136.008, Y  +283.940, Z    +0.000, E1   +73.594, E3 +18423.171}
SPL {X  -132.748, Y  +279.415, Z    +0.000, E1   +73.006, E3 +18429.226}
SPL {X  -129.007, Y  +274.590, Z    +0.000, E1   +72.484, E3 +18434.575}
SPL {X  -124.646, Y  +269.397, Z    +0.000, E1   +72.041, E3 +18439.324}
SPL {X  -111.023, Y  +255.562, Z    +0.000, E1   +75.772, E3 +18431.105}
SPL {X   -52.752, Y  +221.474, Z    +0.000, E1   +59.157, E3 +18560.357}
SPL {X   -49.901, Y  +220.545, Z    +0.000, E1   +56.696, E3 +18646.749}
ENDSPLINE

SPLINE
SPL {X  -127.117, Y  +272.287, Z    +0.000, E1   +62.713, E3 +18793.042}
SPL {X  -152.442, Y  +313.682, Z    +0.000, E1   +51.943, E3 +18797.274}
SPL {X  -159.925, Y  +335.326, Z    +0.000, E1   +41.361, E3 +18797.216}
SPL {X  -163.450, Y  +351.595, Z    +0.000, E1   +29.785, E3 +18796.327}
SPL {X  -165.127, Y  +365.342, Z    +0.000, E1   +17.250, E3 +18796.307}
SPL {X  -165.640, Y  +376.693, Z    +0.000, E1    +4.721, E3 +18795.880}
SPL {X  -165.650, Y  +380.500, Z    +0.000, E1    -0.000, E3 +18795.031}
SPL {X  -165.650, Y  +383.262, Z    +0.000, E1    -6.645, E3 +18794.560}
SPL {X  -165.650, Y  +388.390, Z    +0.000, E1   -21.508, E3 +18794.348}
SPL {X  -165.650, Y  +393.439, Z    +0.000, E1   -35.398, E3 +18793.915}
SPL {X  -165.650, Y  +400.610, Z    +0.000, E1   -50.510, E3 +18793.653}
SPL {X  -165.650, Y  +414.376, Z    +0.000, E1   -68.098, E3 +18791.687}
SPL {X  -165.650, Y  +468.582, Z    +0.000, E1   -78.237, E3 +18800.457}
SPL {X  -158.306, Y  +724.277, Z    +0.000, E1   -77.461, E3 +18890.898}
ENDSPLINE

SPLINE
SPL {X  -160.145, Y  +717.851, Z    +0.000, E1   -75.386, E3 +18911.412}
ENDSPLINE

SPLINE
SPL {X  -157.156, Y  +727.862, Z    +0.000, E1   -75.175, E3 +18918.884}
SPL {X  -152.814, Y  +739.436, Z    +0.000, E1   -74.813, E3 +18928.737}
SPL {X  -147.104, Y  +751.659, Z    +0.000, E1   -74.255, E3 +18940.182}
SPL {X  -141.453, Y  +761.704, Z    +0.000, E1   -73.638, E3 +18950.395}
SPL {X  -135.914, Y  +770.196, Z    +0.000, E1   -72.974, E3 +18959.456}
SPL {X  -131.459, Y  +776.289, Z    +0.000, E1   -72.475, E3 +18965.532}
SPL {X  -127.605, Y  +781.126, Z    +0.000, E1   -71.922, E3 +18970.976}
SPL {X  -124.773, Y  +784.457, Z    +0.000, E1   -71.383, E3 +18975.024}
SPL {X  -119.086, Y  +790.645, Z    +0.000, E1   -72.931, E3 +18971.878}
SPL {X   -51.449, Y  +832.958, Z    +0.000, E1   -57.230, E3 +19129.398}
ENDSPLINE

SPLINE
SPL {X  -123.821, Y  +785.537, Z    +0.000, E1   -64.536, E3 +19331.143}
SPL {X  -153.467, Y  +737.853, Z    +0.000, E1   -51.757, E3 +19333.458}
SPL {X  -162.176, Y  +709.248, Z    +0.000, E1   -35.773, E3 +19332.483}
SPL {X  -164.888, Y  +691.368, Z    +0.000, E1   -20.174, E3 +19330.921}
SPL {X  -165.597, Y  +679.703, Z    +0.000, E1    -7.645, E3 +19331.096}
SPL {X  -165.650, Y  +673.520, Z    +0.000, E1    -0.048, E3 +19330.048}
SPL {X  -165.650, Y  +671.692, Z    +0.000, E1    +4.450, E3 +19329.614}
SPL {X  -165.650, Y  +667.743, Z    +0.000, E1   +15.617, E3 +19329.532}
SPL {X  -165.650, Y  +661.459, Z    +0.000, E1   +33.218, E3 +19329.112}
SPL {X  -165.650, Y  +653.296, Z    +0.000, E1   +51.333, E3 +19328.668}
SPL {X  -165.650, Y  +642.000, Z    +0.000, E1   +65.561, E3 +19327.880}
SPL {X  -165.650, Y  +619.979, Z    +0.000, E1   +79.465, E3 +19323.886}
SPL {X  -165.650, Y  +584.722, Z    +0.000, E1   +79.551, E3 +19333.177}
SPL {X  -165.650, Y  +560.326, Z    +0.000, E1   +78.360, E3 +19342.900}
SPL {X  -160.258, Y  +336.579, Z    +0.000, E1   +78.314, E3 +19414.422}
SPL {X  -159.618, Y  +334.207, Z    +0.000, E1   +75.622, E3 +19445.235}
SPL {X  -157.855, Y  +328.284, Z    +0.000, E1   +75.167, E3 +19453.201}
SPL {X  -155.139, Y  +320.432, Z    +0.000, E1   +75.106, E3 +19457.878}
SPL {X  -142.256, Y  +293.629, Z    +0.000, E1   +77.020, E3 +19450.691}
ENDSPLINE

SPLINE
SPL {X  -142.811, Y  +294.566, Z    +0.000, E1   +75.668, E3 +19462.653}
ENDSPLINE

SPLINE
SPL {X  -141.646, Y  +292.615, Z    +0.000, E1   +74.702, E3 +19471.747}
SPL {X  -140.419, Y  +290.622, Z    +0.000, E1   +73.705, E3 +19480.590}
SPL {X  -136.008, Y  +283.940, Z    +0.000, E1   +73.594, E3 +19484.709}
SPL {X  -131.988, Y  +278.404, Z    +0.000, E1   +72.860, E3 +19492.264}
SPL {X  -126.848, Y  +271.966, Z    +0.000, E1   +72.322, E3 +19498.309}
SPL {X  -123.729, Y  +268.359, Z    +0.000, E1   +71.932, E3 +19501.778}
SPL {X  -111.023, Y  +255.562, Z    +0.000, E1   +75.772, E3 +19492.644}
SPL {X   -49.289, Y  +220.353, Z    +0.000, E1   +56.690, E3 +19685.358}
ENDSPLINE

SPLINE
SPL {X  -127.117, Y  +272.287, Z    +0.000, E1   +62.713, E3 +19854.580}
SPL {X  -152.442, Y  +313.682, Z    +0.000, E1   +51.943, E3 +19858.812}
SPL {X  -159.925, Y  +335.326, Z    +0.000, E1   +41.361, E3 +19858.754}
SPL {X  -163.450, Y  +351.595, Z    +0.000, E1   +29.785, E3 +19857.865}
SPL {X  -165.127, Y  +365.342, Z    +0.000, E1   +17.250, E3 +19857.846}
SPL {X  -165.640, Y  +376.693, Z    +0.000, E1    +4.721, E3 +19857.419}
SPL {X  -165.650, Y  +380.500, Z    +0.000, E1    -0.000, E3 +19856.569}
SPL {X  -165.650, Y  +382.123, Z    +0.000, E1    -3.912, E3 +19856.197}
SPL {X  -165.650, Y  +387.069, Z    +0.000, E1   -17.420, E3 +19855.908}
SPL {X  -165.650, Y  +393.439, Z    +0.000, E1   -35.398, E3 +19855.454}
SPL {X  -165.650, Y  +402.896, Z    +0.000, E1   -54.480, E3 +19854.695}
SPL {X  -165.650, Y  +416.934, Z    +0.000, E1   -69.887, E3 +19853.161}
SPL {X  -165.650, Y  +459.729, Z    +0.000, E1   -78.035, E3 +19859.680}
SPL {X  -165.650, Y  +475.450, Z    +0.000, E1   -78.345, E3 +19863.794}
SPL {X  -158.306, Y  +724.277, Z    +0.000, E1   -77.461, E3 +19952.437}
ENDSPLINE

SPLINE
SPL {X  -160.145, Y  +717.851, Z    +0.000, E1   -75.386, E3 +19972.950}
ENDSPLINE

SPLINE
SPL {X  -157.156, Y  +727.862, Z    +0.000, E1   -75.175, E3 +19980.422}
SPL {X  -154.068, Y  +736.353, Z    +0.000, E1   -74.906, E3 +19987.597}
SPL {X  -149.738, Y  +746.340, Z    +0.000, E1   -74.451, E3 +19997.284}
SPL {X  -145.204, Y  +755.223, Z    +0.000, E1   -74.188, E3 +20004.011}
SPL {X  -141.453, Y  +761.704, Z    +0.000, E1   -73.638, E3 +20011.933}
SPL {X  -135.914, Y  +770.196, Z    +0.000, E1   -72.974, E3 +20020.995}
SPL {X  -131.459, Y  +776.289, Z    +0.000, E1   -72.475, E3 +20027.070}
SPL {X  -128.771, Y  +779.702, Z    +0.000, E1   -71.875, E3 +20032.017}
SPL {X  -124.506, Y  +784.762, Z    +0.000, E1   -71.815, E3 +20034.906}
SPL {X  -112.958, Y  +796.663, Z    +0.000, E1   -74.119, E3 +20031.609}
SPL {X   -51.449, Y  +832.958, Z    +0.000, E1   -57.230, E3 +20190.936}
ENDSPLINE

SPLINE
SPL {X  -123.821, Y  +785.537, Z    +0.000, E1   -64.536, E3 +20392.681}
SPL {X  -153.467, Y  +737.853, Z    +0.000, E1   -51.757, E3 +20394.996}
SPL {X  -162.176, Y  +709.248, Z    +0.000, E1   -35.773, E3 +20394.022}
SPL {X  -164.888, Y  +691.368, Z    +0.000, E1   -20.174, E3 +20392.459}
SPL {X  -165.597, Y  +679.703, Z    +0.000, E1    -7.645, E3 +20392.634}
SPL {X  -165.650, Y  +673.520, Z    +0.000, E1    -0.048, E3 +20391.586}
SPL {X  -165.650, Y  +671.692, Z    +0.000, E1    +4.450, E3 +20391.153}
SPL {X  -165.650, Y  +667.743, Z    +0.000, E1   +15.617, E3 +20391.070}
SPL {X  -165.650, Y  +661.459, Z    +0.000, E1   +33.218, E3 +20390.651}
SPL {X  -165.650, Y  +653.296, Z    +0.000, E1   +51.333, E3 +20390.206}
SPL {X  -165.650, Y  +642.000, Z    +0.000, E1   +65.561, E3 +20389.418}
SPL {X  -165.650, Y  +619.979, Z    +0.000, E1   +79.465, E3 +20385.425}
SPL {X  -165.650, Y  +569.632, Z    +0.000, E1   +78.783, E3 +20400.704}
SPL {X  -158.840, Y  +331.491, Z    +0.000, E1   +77.462, E3 +20487.014}
ENDSPLINE

SPLINE
SPL {X  -159.893, Y  +335.208, Z    +0.000, E1   +75.483, E3 +20507.748}
ENDSPLINE

SPLINE
SPL {X  -156.487, Y  +324.170, Z    +0.000, E1   +75.150, E3 +20517.130}
SPL {X  -142.256, Y  +293.629, Z    +0.000, E1   +77.020, E3 +20512.229}
ENDSPLINE

SPLINE
SPL {X  -142.811, Y  +294.566, Z    +0.000, E1   +75.668, E3 +20524.192}
ENDSPLINE

SPLINE
SPL {X  -141.646, Y  +292.615, Z    +0.000, E1   +74.702, E3 +20533.285}
SPL {X  -140.419, Y  +290.622, Z    +0.000, E1   +73.705, E3 +20542.129}
SPL {X  -135.839, Y  +283.697, Z    +0.000, E1   +73.388, E3 +20547.867}
SPL {X  -131.336, Y  +277.551, Z    +0.000, E1   +72.879, E3 +20554.119}
SPL {X  -126.848, Y  +271.966, Z    +0.000, E1   +72.322, E3 +20559.847}
SPL {X  -123.729, Y  +268.359, Z    +0.000, E1   +71.932, E3 +20563.316}
SPL {X  -111.023, Y  +255.562, Z    +0.000, E1   +75.772, E3 +20554.182}
SPL {X   -52.752, Y  +221.474, Z    +0.000, E1   +59.157, E3 +20683.434}
SPL {X   -49.901, Y  +220.545, Z    +0.000, E1   +56.696, E3 +20769.826}
ENDSPLINE

SPLINE
SPL {X  -127.117, Y  +272.287, Z    +0.000, E1   +62.713, E3 +20916.119}
SPL {X  -152.442, Y  +313.682, Z    +0.000, E1   +51.943, E3 +20920.351}
SPL {X  -162.319, Y  +345.447, Z    +0.000, E1   +34.671, E3 +20919.776}
SPL {X  -165.127, Y  +365.342, Z    +0.000, E1   +17.250, E3 +20919.384}
SPL {X  -165.640, Y  +376.693, Z    +0.000, E1    +4.721, E3 +20918.957}
SPL {X  -165.650, Y  +380.500, Z    +0.000, E1    -0.000, E3 +20918.108}
SPL {X  -165.650, Y  +382.123, Z    +0.000, E1    -3.912, E3 +20917.735}
SPL {X  -165.650, Y  +387.069, Z    +0.000, E1   -17.420, E3 +20917.447}
SPL {X  -165.650, Y  +393.439, Z    +0.000, E1   -35.398, E3 +20916.992}
SPL {X  -165.650, Y  +400.610, Z    +0.000, E1   -50.510, E3 +20916.730}
SPL {X  -165.650, Y  +414.376, Z    +0.000, E1   -68.098, E3 +20914.764}
SPL {X  -165.650, Y  +468.582, Z    +0.000, E1   -78.237, E3 +20923.534}
SPL {X  -160.244, Y  +717.475, Z    +0.000, E1   -78.917, E3 +20996.092}
SPL {X  -159.651, Y  +719.676, Z    +0.000, E1   -75.661, E3 +21032.478}
SPL {X  -157.156, Y  +727.862, Z    +0.000, E1   -75.175, E3 +21041.961}
SPL {X  -154.068, Y  +736.353, Z    +0.000, E1   -74.906, E3 +21049.135}
SPL {X  -149.738, Y  +746.340, Z    +0.000, E1   -74.451, E3 +21058.823}
SPL {X  -144.163, Y  +757.090, Z    +0.000, E1   -74.033, E3 +21067.915}
SPL {X  -139.284, Y  +765.165, Z    +0.000, E1   -73.322, E3 +21077.610}
SPL {X  -134.662, Y  +771.969, Z    +0.000, E1   -72.884, E3 +21083.942}
SPL {X  -131.459, Y  +776.289, Z    +0.000, E1   -72.475, E3 +21088.609}
SPL {X  -127.605, Y  +781.126, Z    +0.000, E1   -71.922, E3 +21094.053}
SPL {X  -124.773, Y  +784.457, Z    +0.000, E1   -71.383, E3 +21098.100}
SPL {X  -119.086, Y  +790.645, Z    +0.000, E1   -72.931, E3 +21094.955}
SPL {X   -51.449, Y  +832.958, Z    +0.000, E1   -57.230, E3 +21252.475}
ENDSPLINE

SPLINE
SPL {X  -123.821, Y  +785.537, Z    +0.000, E1   -64.536, E3 +21454.220}
SPL {X  -153.467, Y  +737.853, Z    +0.000, E1   -51.757, E3 +21456.534}
SPL {X  -161.000, Y  +714.475, Z    +0.000, E1   -39.424, E3 +21456.007}
SPL {X  -164.534, Y  +694.695, Z    +0.000, E1   -23.511, E3 +21454.297}
SPL {X  -165.597, Y  +679.703, Z    +0.000, E1    -7.645, E3 +21454.173}
SPL {X  -165.650, Y  +673.520, Z    +0.000, E1    -0.048, E3 +21453.124}
SPL {X  -165.650, Y  +671.692, Z    +0.000, E1    +4.450, E3 +21452.691}
SPL {X  -165.650, Y  +667.743, Z    +0.000, E1   +15.617, E3 +21452.609}
SPL {X  -165.650, Y  +661.459, Z    +0.000, E1   +33.218, E3 +21452.189}
SPL {X  -165.650, Y  +653.296, Z    +0.000, E1   +51.333, E3 +21451.745}
SPL {X  -165.650, Y  +642.000, Z    +0.000, E1   +65.561, E3 +21450.957}
SPL {X  -165.650, Y  +619.979, Z    +0.000, E1   +79.465, E3 +21446.963}
SPL {X  -165.650, Y  +569.632, Z    +0.000, E1   +78.783, E3 +21462.242}
SPL {X  -158.840, Y  +331.491, Z    +0.000, E1   +77.462, E3 +21548.552}
ENDSPLINE

SPLINE
SPL {X  -159.893, Y  +335.208, Z    +0.000, E1   +75.483, E3 +21569.287}
ENDSPLINE

SPLINE
SPL {X  -156.487, Y  +324.170, Z    +0.000, E1   +75.150, E3 +21578.668}
SPL {X  -142.256, Y  +293.629, Z    +0.000, E1   +77.020, E3 +21573.768}
ENDSPLINE

SPLINE
SPL {X  -142.811, Y  +294.566, Z    +0.000, E1   +75.668, E3 +21585.730}
ENDSPLINE

SPLINE
SPL {X  -141.646, Y  +292.615, Z    +0.000, E1   +74.702, E3 +21594.824}
SPL {X  -140.419, Y  +290.622, Z    +0.000, E1   +73.705, E3 +21603.667}
SPL {X  -136.008, Y  +283.940, Z    +0.000, E1   +73.594, E3 +21607.786}
SPL {X  -132.748, Y  +279.415, Z    +0.000, E1   +73.006, E3 +21613.842}
SPL {X  -129.007, Y  +274.590, Z    +0.000, E1   +72.484, E3 +21619.191}
SPL {X  -125.914, Y  +270.864, Z    +0.000, E1   +72.144, E3 +21622.682}
SPL {X  -123.729, Y  +268.359, Z    +0.000, E1   +71.932, E3 +21624.855}
SPL {X  -111.023, Y  +255.562, Z    +0.000, E1   +75.772, E3 +21615.720}
SPL {X   -49.289, Y  +220.353, Z    +0.000, E1   +56.690, E3 +21808.435}
ENDSPLINE

SPLINE
SPL {X  -127.117, Y  +272.287, Z    +0.000, E1   +62.713, E3 +21977.657}
SPL {X  -154.956, Y  +319.945, Z    +0.000, E1   +49.402, E3 +21982.056}
SPL {X  -162.871, Y  +348.286, Z    +0.000, E1   +32.462, E3 +21981.084}
SPL {X  -165.127, Y  +365.342, Z    +0.000, E1   +17.250, E3 +21980.923}
SPL {X  -165.640, Y  +376.693, Z    +0.000, E1    +4.721, E3 +21980.496}
SPL {X  -165.650, Y  +380.500, Z    +0.000, E1    -0.000, E3 +21979.646}
SPL {X  -165.650, Y  +383.262, Z    +0.000, E1    -6.645, E3 +21979.176}
SPL {X  -165.650, Y  +388.390, Z    +0.000, E1   -21.508, E3 +21978.963}
SPL {X  -165.650, Y  +393.439, Z    +0.000, E1   -35.398, E3 +21978.531}
SPL {X  -165.650, Y  +400.610, Z    +0.000, E1   -50.510, E3 +21978.268}
SPL {X  -165.650, Y  +414.376, Z    +0.000, E1   -68.098, E3 +21976.302}
SPL {X  -165.650, Y  +468.582, Z    +0.000, E1   -78.237, E3 +21985.072}
SPL {X  -158.306, Y  +724.277, Z    +0.000, E1   -77.461, E3 +22075.514}
ENDSPLINE

SPLINE
SPL {X  -160.145, Y  +717.851, Z    +0.000, E1   -75.386, E3 +22096.027}
ENDSPLINE

SPLINE
SPL {X  -157.156, Y  +727.862, Z    +0.000, E1   -75.175, E3 +22103.499}
SPL {X  -154.068, Y  +736.353, Z    +0.000, E1   -74.906, E3 +22110.674}
SPL {X  -149.738, Y  +746.340, Z    +0.000, E1   -74.451, E3 +22120.361}
SPL {X  -144.163, Y  +757.090, Z    +0.000, E1   -74.033, E3 +22129.454}
SPL {X  -139.284, Y  +765.165, Z    +0.000, E1   -73.322, E3 +22139.149}
SPL {X  -134.662, Y  +771.969, Z    +0.000, E1   -72.884, E3 +22145.480}
SPL {X  -131.459, Y  +776.289, Z    +0.000, E1   -72.475, E3 +22150.147}
SPL {X  -127.605, Y  +781.126, Z    +0.000, E1   -71.922, E3 +22155.592}
SPL {X  -124.773, Y  +784.457, Z    +0.000, E1   -71.383, E3 +22159.639}
SPL {X  -119.086, Y  +790.645, Z    +0.000, E1   -72.931, E3 +22156.493}
SPL {X   -51.449, Y  +832.958, Z    +0.000, E1   -57.230, E3 +22314.013}
ENDSPLINE

SPLINE
SPL {X  -123.821, Y  +785.537, Z    +0.000, E1   -64.536, E3 +22515.758}
SPL {X  -153.467, Y  +737.853, Z    +0.000, E1   -51.757, E3 +22518.073}
SPL {X  -161.000, Y  +714.475, Z    +0.000, E1   -39.424, E3 +22517.546}
SPL {X  -164.534, Y  +694.695, Z    +0.000, E1   -23.511, E3 +22515.835}
SPL {X  -165.597, Y  +679.703, Z    +0.000, E1    -7.645, E3 +22515.711}
SPL {X  -165.650, Y  +673.520, Z    +0.000, E1    -0.048, E3 +22514.663}
SPL {X  -165.650, Y  +671.692, Z    +0.000, E1    +4.450, E3 +22514.230}
SPL {X  -165.650, Y  +667.743, Z    +0.000, E1   +15.617, E3 +22514.147}
SPL {X  -165.650, Y  +661.459, Z    +0.000, E1   +33.218, E3 +22513.728}
SPL {X  -165.650, Y  +653.296, Z    +0.000, E1   +51.333, E3 +22513.283}
SPL {X  -165.650, Y  +642.000, Z    +0.000, E1   +65.561, E3 +22512.495}
SPL {X  -165.650, Y  +619.979, Z    +0.000, E1   +79.465, E3 +22508.502}
SPL {X  -165.650, Y  +569.632, Z    +0.000, E1   +78.783, E3 +22523.781}
SPL {X  -158.840, Y  +331.491, Z    +0.000, E1   +77.462, E3 +22610.091}
ENDSPLINE

SPLINE
SPL {X  -159.893, Y  +335.208, Z    +0.000, E1   +75.483, E3 +22630.825}
ENDSPLINE

SPLINE
SPL {X  -156.487, Y  +324.170, Z    +0.000, E1   +75.150, E3 +22640.207}
SPL {X  -142.256, Y  +293.629, Z    +0.000, E1   +77.020, E3 +22635.306}
ENDSPLINE

SPLINE
SPL {X  -142.811, Y  +294.566, Z    +0.000, E1   +75.668, E3 +22647.269}
ENDSPLINE

SPLINE
SPL {X  -141.646, Y  +292.615, Z    +0.000, E1   +74.702, E3 +22656.362}
SPL {X  -140.419, Y  +290.622, Z    +0.000, E1   +73.705, E3 +22665.205}
SPL {X  -136.008, Y  +283.940, Z    +0.000, E1   +73.594, E3 +22669.325}
SPL {X  -132.748, Y  +279.415, Z    +0.000, E1   +73.006, E3 +22675.380}
SPL {X  -129.007, Y  +274.590, Z    +0.000, E1   +72.484, E3 +22680.729}
SPL {X  -125.914, Y  +270.864, Z    +0.000, E1   +72.144, E3 +22684.221}
SPL {X  -123.729, Y  +268.359, Z    +0.000, E1   +71.932, E3 +22686.393}
SPL {X  -111.023, Y  +255.562, Z    +0.000, E1   +75.772, E3 +22677.259}
SPL {X   -49.289, Y  +220.353, Z    +0.000, E1   +56.690, E3 +22869.974}
ENDSPLINE

SPLINE
SPL {X  -127.117, Y  +272.287, Z    +0.000, E1   +62.713, E3 +23039.196}
SPL {X  -152.442, Y  +313.682, Z    +0.000, E1   +51.943, E3 +23043.428}
SPL {X  -162.319, Y  +345.447, Z    +0.000, E1   +34.671, E3 +23042.853}
SPL {X  -165.127, Y  +365.342, Z    +0.000, E1   +17.250, E3 +23042.461}
SPL {X  -165.640, Y  +376.693, Z    +0.000, E1    +4.721, E3 +23042.034}
SPL {X  -165.650, Y  +380.500, Z    +0.000, E1    -0.000, E3 +23041.185}
SPL {X  -165.650, Y  +383.262, Z    +0.000, E1    -6.645, E3 +23040.714}
SPL {X  -165.650, Y  +388.390, Z    +0.000, E1   -21.508, E3 +23040.502}
SPL {X  -165.650, Y  +393.439, Z    +0.000, E1   -35.398, E3 +23040.069}
SPL {X  -165.650, Y  +400.610, Z    +0.000, E1   -50.510, E3 +23039.807}
SPL {X  -165.650, Y  +414.376, Z    +0.000, E1   -68.098, E3 +23037.841}
SPL {X  -165.650, Y  +468.582, Z    +0.000, E1   -78.237, E3 +23046.611}
SPL {X  -158.306, Y  +724.277, Z    +0.000, E1   -77.461, E3 +23137.052}
ENDSPLINE

SPLINE
SPL {X  -160.145, Y  +717.851, Z    +0.000, E1   -75.386, E3 +23157.565}
ENDSPLINE

SPLINE
SPL {X  -157.156, Y  +727.862, Z    +0.000, E1   -75.175, E3 +23165.038}
SPL {X  -154.068, Y  +736.353, Z    +0.000, E1   -74.906, E3 +23172.212}
SPL {X  -149.738, Y  +746.340, Z    +0.000, E1   -74.451, E3 +23181.900}
SPL {X  -144.163, Y  +757.090, Z    +0.000, E1   -74.033, E3 +23190.992}
SPL {X  -139.284, Y  +765.165, Z    +0.000, E1   -73.322, E3 +23200.687}
SPL {X  -134.662, Y  +771.969, Z    +0.000, E1   -72.884, E3 +23207.019}
SPL {X  -131.459, Y  +776.289, Z    +0.000, E1   -72.475, E3 +23211.686}
SPL {X  -127.605, Y  +781.126, Z    +0.000, E1   -71.922, E3 +23217.130}
SPL {X  -124.773, Y  +784.457, Z    +0.000, E1   -71.383, E3 +23221.177}
SPL {X  -119.086, Y  +790.645, Z    +0.000, E1   -72.931, E3 +23218.032}
SPL {X   -51.449, Y  +832.958, Z    +0.000, E1   -57.230, E3 +23375.551}
ENDSPLINE

SPLINE
SPL {X  -123.821, Y  +785.537, Z    +0.000, E1   -64.536, E3 +23577.297}
SPL {X  -153.467, Y  +737.853, Z    +0.000, E1   -51.757, E3 +23579.611}
SPL {X  -162.176, Y  +709.248, Z    +0.000, E1   -35.773, E3 +23578.637}
SPL {X  -164.888, Y  +691.368, Z    +0.000, E1   -20.174, E3 +23577.075}
SPL {X  -165.597, Y  +679.703, Z    +0.000, E1    -7.645, E3 +23577.250}
SPL {X  -165.650, Y  +673.520, Z    +0.000, E1    -0.048, E3 +23576.201}
SPL {X  -165.650, Y  +671.692, Z    +0.000, E1    +4.450, E3 +23575.768}
SPL {X  -165.650, Y  +667.743, Z    +0.000, E1   +15.617, E3 +23575.686}
SPL {X  -165.650, Y  +661.459, Z    +0.000, E1   +33.218, E3 +23575.266}
SPL {X  -165.650, Y  +653.296, Z    +0.000, E1   +51.333, E3 +23574.822}
SPL {X  -165.650, Y  +642.000, Z    +0.000, E1   +65.561, E3 +23574.034}
SPL {X  -165.650, Y  +619.979, Z    +0.000, E1   +79.465, E3 +23570.040}
SPL {X  -165.650, Y  +584.722, Z    +0.000, E1   +79.551, E3 +23579.331}
SPL {X  -165.650, Y  +560.326, Z    +0.000, E1   +78.360, E3 +23589.054}
SPL {X  -158.840, Y  +331.491, Z    +0.000, E1   +77.462, E3 +23671.629}
ENDSPLINE

SPLINE
SPL {X  -159.893, Y  +335.208, Z    +0.000, E1   +75.483, E3 +23692.364}
ENDSPLINE

SPLINE
SPL {X  -156.487, Y  +324.170, Z    +0.000, E1   +75.150, E3 +23701.745}
SPL {X  -142.256, Y  +293.629, Z    +0.000, E1   +77.020, E3 +23696.845}
ENDSPLINE

SPLINE
SPL {X  -142.811, Y  +294.566, Z    +0.000, E1   +75.668, E3 +23708.807}
ENDSPLINE

SPLINE
SPL {X  -141.646, Y  +292.615, Z    +0.000, E1   +74.702, E3 +23717.901}
SPL {X  -140.419, Y  +290.622, Z    +0.000, E1   +73.705, E3 +23726.744}
SPL {X  -136.008, Y  +283.940, Z    +0.000, E1   +73.594, E3 +23730.863}
SPL {X  -132.748, Y  +279.415, Z    +0.000, E1   +73.006, E3 +23736.919}
SPL {X  -129.007, Y  +274.590, Z    +0.000, E1   +72.484, E3 +23742.268}
SPL {X  -125.914, Y  +270.864, Z    +0.000, E1   +72.144, E3 +23745.759}
SPL {X  -123.729, Y  +268.359, Z    +0.000, E1   +71.932, E3 +23747.932}
SPL {X  -111.023, Y  +255.562, Z    +0.000, E1   +75.772, E3 +23738.797}
SPL {X   -49.289, Y  +220.353, Z    +0.000, E1   +56.690, E3 +23931.512}
ENDSPLINE

SPLINE
SPL {X  -127.117, Y  +272.287, Z    +0.000, E1   +62.713, E3 +24100.734}
SPL {X  -152.442, Y  +313.682, Z    +0.000, E1   +51.943, E3 +24104.966}
SPL {X  -159.925, Y  +335.326, Z    +0.000, E1   +41.361, E3 +24104.908}
SPL {X  -163.450, Y  +351.595, Z    +0.000, E1   +29.785, E3 +24104.019}
SPL {X  -165.127, Y  +365.342, Z    +0.000, E1   +17.250, E3 +24104.000}
SPL {X  -165.640, Y  +376.693, Z    +0.000, E1    +4.721, E3 +24103.572}
SPL {X  -165.650, Y  +380.500, Z    +0.000, E1    -0.000, E3 +24102.723}
SPL {X  -165.650, Y  +382.123, Z    +0.000, E1    -3.912, E3 +24102.351}
SPL {X  -165.650, Y  +387.069, Z    +0.000, E1   -17.420, E3 +24102.062}
SPL {X  -165.650, Y  +393.439, Z    +0.000, E1   -35.398, E3 +24101.608}
SPL {X  -165.650, Y  +400.610, Z    +0.000, E1   -50.510, E3 +24101.345}
SPL {X  -165.650, Y  +414.376, Z    +0.000, E1   -68.098, E3 +24099.379}
SPL {X  -165.650, Y  +468.582, Z    +0.000, E1   -78.237, E3 +24108.149}
SPL {X  -160.244, Y  +717.475, Z    +0.000, E1   -78.917, E3 +24180.707}
SPL {X  -159.651, Y  +719.676, Z    +0.000, E1   -75.661, E3 +24217.094}
SPL {X  -157.156, Y  +727.862, Z    +0.000, E1   -75.175, E3 +24226.576}
SPL {X  -152.814, Y  +739.436, Z    +0.000, E1   -74.813, E3 +24236.430}
SPL {X  -148.754, Y  +748.385, Z    +0.000, E1   -74.281, E3 +24245.872}
SPL {X  -144.163, Y  +757.090, Z    +0.000, E1   -74.033, E3 +24252.531}
SPL {X  -140.473, Y  +763.291, Z    +0.000, E1   -73.478, E3 +24259.972}
SPL {X  -135.914, Y  +770.196, Z    +0.000, E1   -72.974, E3 +24267.148}
SPL {X  -131.459, Y  +776.289, Z    +0.000, E1   -72.475, E3 +24273.224}
SPL {X  -128.771, Y  +779.702, Z    +0.000, E1   -71.875, E3 +24278.171}
SPL {X  -125.267, Y  +783.889, Z    +0.000, E1   -71.674, E3 +24281.283}
SPL {X  -119.086, Y  +790.645, Z    +0.000, E1   -72.931, E3 +24279.570}
SPL {X   -51.449, Y  +832.958, Z    +0.000, E1   -57.230, E3 +24437.090}
ENDSPLINE

SPLINE
SPL {X  -123.821, Y  +785.537, Z    +0.000, E1   -64.536, E3 +24638.835}
SPL {X  -153.467, Y  +737.853, Z    +0.000, E1   -51.757, E3 +24641.150}
SPL {X  -161.000, Y  +714.475, Z    +0.000, E1   -39.424, E3 +24640.622}
SPL {X  -164.534, Y  +694.695, Z    +0.000, E1   -23.511, E3 +24638.912}
SPL {X  -165.597, Y  +679.703, Z    +0.000, E1    -7.645, E3 +24638.788}
SPL {X  -165.650, Y  +673.520, Z    +0.000, E1    -0.048, E3 +24637.740}
SPL {X  -165.650, Y  +671.692, Z    +0.000, E1    +4.450, E3 +24637.306}
SPL {X  -165.650, Y  +667.743, Z    +0.000, E1   +15.617, E3 +24637.224}
SPL {X  -165.650, Y  +662.891, Z    +0.000, E1   +29.740, E3 +24636.742}
SPL {X  -165.650, Y  +655.319, Z    +0.000, E1   +47.265, E3 +24636.591}
SPL {X  -165.650, Y  +642.000, Z    +0.000, E1   +65.561, E3 +24635.572}
SPL {X  -165.650, Y  +619.979, Z    +0.000, E1   +79.465, E3 +24631.579}
SPL {X  -165.650, Y  +569.632, Z    +0.000, E1   +78.783, E3 +24646.858}
SPL {X  -158.840, Y  +331.491, Z    +0.000, E1   +77.462, E3 +24733.168}
ENDSPLINE

SPLINE
SPL {X  -159.893, Y  +335.208, Z    +0.000, E1   +75.483, E3 +24753.902}
ENDSPLINE

SPLINE
SPL {X  -156.487, Y  +324.170, Z    +0.000, E1   +75.150, E3 +24763.283}
SPL {X  -142.256, Y  +293.629, Z    +0.000, E1   +77.020, E3 +24758.383}
ENDSPLINE

SPLINE
SPL {X  -142.811, Y  +294.566, Z    +0.000, E1   +75.668, E3 +24770.346}
ENDSPLINE

SPLINE
SPL {X  -141.646, Y  +292.615, Z    +0.000, E1   +74.702, E3 +24779.439}
SPL {X  -140.419, Y  +290.622, Z    +0.000, E1   +73.705, E3 +24788.282}
SPL {X  -135.839, Y  +283.697, Z    +0.000, E1   +73.388, E3 +24794.021}
SPL {X  -131.903, Y  +278.292, Z    +0.000, E1   +73.096, E3 +24798.510}
SPL {X  -129.007, Y  +274.590, Z    +0.000, E1   +72.484, E3 +24803.806}
SPL {X  -124.646, Y  +269.397, Z    +0.000, E1   +72.041, E3 +24808.554}
SPL {X  -111.023, Y  +255.562, Z    +0.000, E1   +75.772, E3 +24800.336}
SPL {X   -49.289, Y  +220.353, Z    +0.000, E1   +56.690, E3 +24993.051}
ENDSPLINE

SPLINE
SPL {X  -127.117, Y  +272.287, Z    +0.000, E1   +62.713, E3 +25162.273}
SPL {X  -154.956, Y  +319.945, Z    +0.000, E1   +49.402, E3 +25166.672}
SPL {X  -162.871, Y  +348.286, Z    +0.000, E1   +32.462, E3 +25165.699}
SPL {X  -165.127, Y  +365.342, Z    +0.000, E1   +17.250, E3 +25165.538}
SPL {X  -165.640, Y  +376.693, Z    +0.000, E1    +4.721, E3 +25165.111}
SPL {X  -165.650, Y  +380.500, Z    +0.000, E1    -0.000, E3 +25164.262}
SPL {X  -165.650, Y  +382.123, Z    +0.000, E1    -3.912, E3 +25163.889}
SPL {X  -165.650, Y  +387.069, Z    +0.000, E1   -17.420, E3 +25163.600}
SPL {X  -165.650, Y  +393.439, Z    +0.000, E1   -35.398, E3 +25163.146}
SPL {X  -165.650, Y  +400.610, Z    +0.000, E1   -50.510, E3 +25162.884}
SPL {X  -165.650, Y  +414.376, Z    +0.000, E1   -68.098, E3 +25160.917}
SPL {X  -165.650, Y  +468.582, Z    +0.000, E1   -78.237, E3 +25169.688}
SPL {X  -160.244, Y  +717.475, Z    +0.000, E1   -78.917, E3 +25242.246}
SPL {X  -159.651, Y  +719.676, Z    +0.000, E1   -75.661, E3 +25278.632}
SPL {X  -157.156, Y  +727.862, Z    +0.000, E1   -75.175, E3 +25288.114}
SPL {X  -154.068, Y  +736.353, Z    +0.000, E1   -74.906, E3 +25295.289}
SPL {X  -149.738, Y  +746.340, Z    +0.000, E1   -74.451, E3 +25304.977}
SPL {X  -144.163, Y  +757.090, Z    +0.000, E1   -74.033, E3 +25314.069}
SPL {X  -139.284, Y  +765.165, Z    +0.000, E1   -73.322, E3 +25323.764}
SPL {X  -134.662, Y  +771.969, Z    +0.000, E1   -72.884, E3 +25330.096}
SPL {X  -131.459, Y  +776.289, Z    +0.000, E1   -72.475, E3 +25334.763}
SPL {X  -127.605, Y  +781.126, Z    +0.000, E1   -71.922, E3 +25340.207}
SPL {X  -124.773, Y  +784.457, Z    +0.000, E1   -71.383, E3 +25344.254}
SPL {X  -119.086, Y  +790.645, Z    +0.000, E1   -72.931, E3 +25341.109}
SPL {X   -51.449, Y  +832.958, Z    +0.000, E1   -57.230, E3 +25498.628}
ENDSPLINE

SPLINE
SPL {X  -123.821, Y  +785.537, Z    +0.000, E1   -64.536, E3 +25700.374}
SPL {X  -153.467, Y  +737.853, Z    +0.000, E1   -51.757, E3 +25702.688}
SPL {X  -161.000, Y  +714.475, Z    +0.000, E1   -39.424, E3 +25702.161}
SPL {X  -164.534, Y  +694.695, Z    +0.000, E1   -23.511, E3 +25700.451}
SPL {X  -165.597, Y  +679.703, Z    +0.000, E1    -7.645, E3 +25700.327}
SPL {X  -165.650, Y  +673.520, Z    +0.000, E1    -0.048, E3 +25699.278}
SPL {X  -165.650, Y  +671.692, Z    +0.000, E1    +4.450, E3 +25698.845}
SPL {X  -165.650, Y  +667.743, Z    +0.000, E1   +15.617, E3 +25698.763}
SPL {X  -165.650, Y  +662.891, Z    +0.000, E1   +29.740, E3 +25698.281}
SPL {X  -165.650, Y  +658.373, Z    +0.000, E1   +40.877, E3 +25698.478}
SPL {X  -165.650, Y  +650.834, Z    +0.000, E1   +55.143, E3 +25697.731}
SPL {X  -165.650, Y  +639.785, Z    +0.000, E1   +67.512, E3 +25696.948}
SPL {X  -165.650, Y  +619.979, Z    +0.000, E1   +79.465, E3 +25693.117}
SPL {X  -165.650, Y  +584.722, Z    +0.000, E1   +79.551, E3 +25702.408}
SPL {X  -165.650, Y  +560.326, Z    +0.000, E1   +78.360, E3 +25712.131}
SPL {X  -160.258, Y  +336.579, Z    +0.000, E1   +78.314, E3 +25783.652}
SPL {X  -159.618, Y  +334.207, Z    +0.000, E1   +75.622, E3 +25814.466}
SPL {X  -156.487, Y  +324.170, Z    +0.000, E1   +75.150, E3 +25824.822}
SPL {X  -142.256, Y  +293.629, Z    +0.000, E1   +77.020, E3 +25819.922}
ENDSPLINE

SPLINE
SPL {X  -142.811, Y  +294.566, Z    +0.000, E1   +75.668, E3 +25831.884}
ENDSPLINE

SPLINE
SPL {X  -141.646, Y  +292.615, Z    +0.000, E1   +74.702, E3 +25840.978}
SPL {X  -140.419, Y  +290.622, Z    +0.000, E1   +73.705, E3 +25849.821}
SPL {X  -136.008, Y  +283.940, Z    +0.000, E1   +73.594, E3 +25853.940}
SPL {X  -132.748, Y  +279.415, Z    +0.000, E1   +73.006, E3 +25859.996}
SPL {X  -129.007, Y  +274.590, Z    +0.000, E1   +72.484, E3 +25865.345}
SPL {X  -125.914, Y  +270.864, Z    +0.000, E1   +72.144, E3 +25868.836}
SPL {X  -123.729, Y  +268.359, Z    +0.000, E1   +71.932, E3 +25871.008}
SPL {X  -111.023, Y  +255.562, Z    +0.000, E1   +75.772, E3 +25861.874}
SPL {X   -52.752, Y  +221.474, Z    +0.000, E1   +59.157, E3 +25991.126}
SPL {X   -49.901, Y  +220.545, Z    +0.000, E1   +56.696, E3 +26077.518}
ENDSPLINE

SPLINE
SPL {X  -127.117, Y  +272.287, Z    +0.000, E1   +62.713, E3 +26223.811}
SPL {X  -152.442, Y  +313.682, Z    +0.000, E1   +51.943, E3 +26228.043}
SPL {X  -162.319, Y  +345.447, Z    +0.000, E1   +34.671, E3 +26227.468}
SPL {X  -165.127, Y  +365.342, Z    +0.000, E1   +17.250, E3 +26227.076}
SPL {X  -165.640, Y  +376.693, Z    +0.000, E1    +4.721, E3 +26226.649}
SPL {X  -165.650, Y  +380.500, Z    +0.000, E1    -0.000, E3 +26225.800}
SPL {X  -165.650, Y  +382.123, Z    +0.000, E1    -3.912, E3 +26225.428}
SPL {X  -165.650, Y  +387.069, Z    +0.000, E1   -17.420, E3 +26225.139}
SPL {X  -165.650, Y  +393.439, Z    +0.000, E1   -35.398, E3 +26224.685}
SPL {X  -165.650, Y  +400.610, Z    +0.000, E1   -50.510, E3 +26224.422}
SPL {X  -165.650, Y  +414.376, Z    +0.000, E1   -68.098, E3 +26222.456}
SPL {X  -165.650, Y  +468.582, Z    +0.000, E1   -78.237, E3 +26231.226}
SPL {X  -160.244, Y  +717.475, Z    +0.000, E1   -78.917, E3 +26303.784}
SPL {X  -159.651, Y  +719.676, Z    +0.000, E1   -75.661, E3 +26340.171}
SPL {X  -157.156, Y  +727.862, Z    +0.000, E1   -75.175, E3 +26349.653}
SPL {X  -154.068, Y  +736.353, Z    +0.000, E1   -74.906, E3 +26356.828}
SPL {X  -149.738, Y  +746.340, Z    +0.000, E1   -74.451, E3 +26366.515}
SPL {X  -144.163, Y  +757.090, Z    +0.000, E1   -74.033, E3 +26375.608}
SPL {X  -139.284, Y  +765.165, Z    +0.000, E1   -73.322, E3 +26385.302}
SPL {X  -134.662, Y  +771.969, Z    +0.000, E1   -72.884, E3 +26391.634}
SPL {X  -131.459, Y  +776.289, Z    +0.000, E1   -72.475, E3 +26396.301}
SPL {X  -127.605, Y  +781.126, Z    +0.000, E1   -71.922, E3 +26401.745}
SPL {X  -124.773, Y  +784.457, Z    +0.000, E1   -71.383, E3 +26405.793}
SPL {X  -119.086, Y  +790.645, Z    +0.000, E1   -72.931, E3 +26402.647}
SPL {X   -51.449, Y  +832.958, Z    +0.000, E1   -57.230, E3 +26560.167}
ENDSPLINE

